// TwinCAT 3 PLC project PLC_1
// Title: ProBox
// Company: Swisslog
// Author: .
// ProjectVersion: 1.0.0
// Description: Based on BCF 1.3.0
// ProgramVersion: 3.1.4023.0
// libraries:
//   Tc2_EtherCAT, * (Beckhoff Automation GmbH)
//   Tc2_MC2, * (Beckhoff Automation GmbH)
//   Tc2_MDP, * (Beckhoff Automation GmbH)
//   Tc2_Standard, * (Beckhoff Automation GmbH)
//   Tc2_System, * (Beckhoff Automation GmbH)
//   Tc2_TcpIp, * (Beckhoff Automation GmbH)
//   Tc2_Utilities, * (Beckhoff Automation GmbH)
//   Tc3_Module, * (Beckhoff Automation GmbH)
// project tree:
//   10_Project/10_App/10_Config/00_GVLs/ Groups.TcGVL, GVL_Safety.TcGVL, HardwareMapping.TcGVL, Positions.TcGVL, ProBoxSystem.TcGVL, Subsystem.TcGVL
//   10_Project/10_App/10_Config/01_DUTs/ E_ElementNumber.TcDUT, E_FunctionNumber.TcDUT, E_GroupNumber.TcDUT
//   10_Project/10_App/10_Config/ F_ConfigCommunication.TcPOU, F_ConfigExternalDestination.TcPOU, F_ConfigGroup.TcPOU, F_ConfigGroupManager.TcPOU, F_ConfigPosition.TcPOU, F_ConfigPosition_001.TcPOU, F_ConfigPosition_002.TcPOU, F_ConfigProduct.TcPOU, F_ConfigSubSystem.TcPOU, F_UpdateISR.TcPOU, F_UpdateReferences.TcPOU
//   10_Project/10_App/11_Custom/ FB_ElementCompositionCustomized.TcPOU, FB_FunctionCompositionCustomized.TcPOU, FB_GroupCompositionCustomized.TcPOU, FB_HardwareInputs.TcPOU, FB_HardwareOutputs.TcPOU, FB_SafetyCompositionCustomized.TcPOU, FB_SubsystemCompositionCustomized.TcPOU, F_DebugCompositionCustomization.TcPOU
//   10_Project/10_App/12_FlowControl/00_GVLs/ FlowControl.TcGVL
//   10_Project/10_App/12_FlowControl/ FB_MergingService.TcPOU, FB_MergingService_001.TcPOU, FB_RoutingService.TcPOU, FB_RoutingService_001.TcPOU
//   10_Project/11_Emu/10_Config/00_GVLs/ GroupsEmulation.TcGVL, PositionsEmulation.TcGVL, SubsystemEmulation.TcGVL
//   10_Project/11_Emu/10_Config/ F_ConfigCommunicationEmulation.TcPOU, F_ConfigGroupEmulation.TcPOU, F_ConfigPositionEmulation.TcPOU, F_ConfigPositionEmulation_001.TcPOU, F_ConfigPositionEmulation_002.TcPOU, F_ConfigProductEmulation.TcPOU, F_ConfigSubSystemEmulation.TcPOU, F_UpdateReferencesEmulation.TcPOU
//   20_Product/10_BCF/10_Base/00_GVLs/ GVR_Table.TcGVL, ISR_Table.TcGVL, RegistryEmulation.TcGVL, SDI_Table.TcGVL, SDO_Table.TcGVL, System.TcGVL, SystemEmulation.TcGVL
//   20_Product/10_BCF/10_Base/01_DUTs/ E_CM_Index.TcDUT, E_CM_Mode.TcDUT, E_ErrorState.TcDUT, E_ErrorType.TcDUT, E_MFCS_Channel.TcDUT, E_PositionMode.TcDUT, E_PositionState.TcDUT, ST_Base.TcDUT, ST_CM_Base.TcDUT, ST_CM_GeneralData.TcDUT, ST_CM_Log.TcDUT, ST_CM_Settings.TcDUT, ST_ISR_Table.TcDUT, ST_PointerSet.TcDUT, ST_PositionInfo.TcDUT, ST_PositionState.TcDUT, ST_SDI_Table.TcDUT, ST_VIR_Data.TcDUT
//   20_Product/10_BCF/10_Base/10_StateMachine/ A_InstancePath.TcDUT, A_StateText.TcDUT, FB_StateMachine.TcPOU, I_StateMachineTextCallback.TcIO
//   20_Product/10_BCF/10_Base/11_Com/01_Stringhandling/ F_InstancePathRemovals.TcPOU, F_StringCopy.TcPOU, F_StringFromDatestruct.TcPOU, F_StringFromTime.TcPOU, F_StringFromTimestruct.TcPOU, F_StringFromUlint.TcPOU, F_StringFromWord.TcPOU, F_StringToTimeDate.TcPOU
//   20_Product/10_BCF/10_Base/11_Com/02_Timings/ E_BlinkFrequencies.TcDUT, F_GetBlinkCycle.TcPOU, F_GetTimeMsDiff.TcPOU, F_GetTimeMsTick.TcPOU, F_GetTimeRemain.TcPOU
//   20_Product/10_BCF/10_Base/11_Com/12_DebugMsg/00_GVLs/ DebugTextBlocks.TcGVL
//   20_Product/10_BCF/10_Base/11_Com/12_DebugMsg/01_DUTs/ E_DebugMsgType.TcDUT, ST_CFG_DebugMsgManager.TcDUT
//   20_Product/10_BCF/10_Base/11_Com/12_DebugMsg/20_TraceHandler/ FB_TraceHandler.TcPOU, I_TraceHandler.TcIO
//   20_Product/10_BCF/10_Base/11_Com/12_DebugMsg/20_TraceHandler/_internal/ A_TracePath.TcDUT (not stored)
//   20_Product/10_BCF/10_Base/11_Com/12_DebugMsg/20_TraceHandler/_internal/entry/ FB_TraceEntry.TcPOU (not stored)
//   20_Product/10_BCF/10_Base/11_Com/12_DebugMsg/20_TraceHandler/_internal/hdd_monitor/ E_ReadHddUsageStates.TcDUT (not stored), FB_HddUsage.TcPOU (not stored), F_DiskSpaceToString.TcPOU (not stored), I_HddUsage.TcIO (not stored)
//   20_Product/10_BCF/10_Base/11_Com/12_DebugMsg/20_TraceHandler/_internal/states/ E_TraceCheckStates.TcDUT (not stored), E_TraceDeleteStates.TcDUT (not stored), E_TraceHddUsageStates.TcDUT (not stored), E_TraceWriteStates.TcDUT (not stored)
//   20_Product/10_BCF/10_Base/11_Com/12_DebugMsg/20_TraceHandler/_internal/statistics/ FB_TraceHandlerStatistics.TcPOU (not stored), I_TraceHandlerStatistics.TcIO (not stored)
//   20_Product/10_BCF/10_Base/11_Com/12_DebugMsg/ FB_DebugMsg.TcPOU, FB_DebugMsgManager.TcPOU
//   20_Product/10_BCF/10_Base/11_Com/ F_InitializeCommunication.TcPOU, F_ITC_SendVIR.TcPOU, ITF_ITC.TcIO, ITF_MFCS.TcIO, ITF_MFCS_Emulation.TcIO
//   20_Product/10_BCF/10_Base/ FB_BaseObject.TcPOU, FB_BaseObjectEmulation.TcPOU, F_ExecutionTime.TcPOU, F_MemStringReplace.TcPOU
//   20_Product/10_BCF/11_Conv/09_Emulation/ MainConvEmulation.TcPOU
//   20_Product/10_BCF/11_Conv/10_Base/00_GVLs/ Conveyor.TcGVL, ExecutionTimeTable.TcGVL, Registry.TcGVL, TU_Table.TcGVL
//   20_Product/10_BCF/11_Conv/10_Base/01_DUTs/ E_ErrorConv.TcDUT, E_EtherCAT_MasterError.TcDUT, ST_ControlRequest.TcDUT, ST_DataSet.TcDUT, ST_DataSetEmulation.TcDUT, ST_Dimension.TcDUT, ST_ElementRegistryConv.TcDUT, ST_ElementRegistryConvEmulation.TcDUT, ST_ErrorDataSet.TcDUT, ST_EtherCATDeviceStates.TcDUT, ST_ExecutionTime.TcDUT, ST_ExternalDestination.TcDUT, ST_FunctionRegistryConv.TcDUT, ST_FunctionRegistryConvEmulation.TcDUT, ST_GroupRegistryConv.TcDUT, ST_GroupRegistryConvEmulation.TcDUT, ST_InitRelease.TcDUT, ST_Interlock.TcDUT, ST_Label.TcDUT, ST_LabelEmulation.TcDUT, ST_PositionIdent.TcDUT, ST_Profile.TcDUT, ST_SubSystemRegistryConv.TcDUT, ST_SubsystemRegistryConvEmulation.TcDUT, ST_TimeStamp.TcDUT, ST_TU_Data.TcDUT, ST_TU_DataEmulation.TcDUT, ST_TU_ID.TcDUT, ST_ZoneRegistryConv.TcDUT, U_ErrorCode.TcDUT
//   20_Product/10_BCF/11_Conv/10_Base/13_GroupManager/01_DUTs/ ST_CFG_GroupManager.TcDUT
//   20_Product/10_BCF/11_Conv/10_Base/13_GroupManager/ FB_GroupManager.TcPOU
//   20_Product/10_BCF/11_Conv/10_Base/ ConveyorEmulation.TcGVL, FB_CommunicationComposition.TcPOU, FB_CommunicationCompositionEmulation.TcPOU, FB_DeleteOldTU_Data.TcPOU, FB_ElementComposition.TcPOU, FB_ElementCompositionEmulation.TcPOU, FB_FunctionComposition.TcPOU, FB_FunctionCompositionEmulation.TcPOU, FB_GroupComposition.TcPOU, FB_GroupCompositionEmulation.TcPOU, FB_SubSystemComposition.TcPOU, FB_SubSystemCompositionEmulation.TcPOU, F_DeleteDestination.TcPOU, F_DeleteTU_Data.TcPOU, F_GetTU_DataIndex.TcPOU, F_GetVirtualDestination.TcPOU, F_InsertTU_Data.TcPOU, F_MonitorEtherCAT_Master.TcPOU, F_ResetError.TcPOU, F_SearchAssignmentId.TcPOU, F_SearchPositionOfTU_Index.TcPOU, F_SearchTU_ByHashCode.TcPOU, F_SetError.TcPOU
//   20_Product/10_BCF/11_Conv/11_Com/11_ITC/01_DUTs/ E_ITC_MsgTypeConv.TcDUT, ST_CFG_ITC_ManagerConv.TcDUT, ST_ITC_ADD_TU_DATA.TcDUT, ST_ITC_ATQ.TcDUT, ST_ITC_ATR.TcDUT, ST_ITC_DAQ.TcDUT, ST_ITC_DAR.TcDUT, ST_ITC_DIQ.TcDUT, ST_ITC_ECQ.TcDUT, ST_ITC_ECR.TcDUT, ST_ITC_ERQ.TcDUT, ST_ITC_ERR.TcDUT, ST_ITC_ESQ.TcDUT, ST_ITC_ESR.TcDUT, ST_ITC_FCQ.TcDUT, ST_ITC_FCR.TcDUT, ST_ITC_FSQ.TcDUT, ST_ITC_FSR.TcDUT, ST_ITC_GCQ.TcDUT, ST_ITC_GCR.TcDUT, ST_ITC_GDQ.TcDUT, ST_ITC_GDR.TcDUT, ST_ITC_GeneralData.TcDUT (not stored), ST_ITC_GSQ.TcDUT (not stored), ST_ITC_GSR.TcDUT (not stored), ST_ITC_GVQ.TcDUT (not stored), ST_ITC_GVR.TcDUT (not stored), ST_ITC_IPR.TcDUT (not stored), ST_ITC_IRQ.TcDUT (not stored), ST_ITC_ISR.TcDUT (not stored), ST_ITC_ManualMotion.TcDUT (not stored), ST_ITC_ManualMotionAxis.TcDUT (not stored), ST_ITC_ManualMotionSelection.TcDUT (not stored), ST_ITC_ManualMotionSpeed.TcDUT (not stored), ST_ITC_MCQ.TcDUT (not stored), ST_ITC_MCR.TcDUT (not stored), ST_ITC_POR.TcDUT (not stored), ST_ITC_RAA.TcDUT (not stored), ST_ITC_RAA_CommandArgs.TcDUT (not stored), ST_ITC_RAC.TcDUT (not stored), ST_ITC_RAQ.TcDUT (not stored), ST_ITC_RDQ.TcDUT (not stored), ST_ITC_RDR.TcDUT (not stored), ST_ITC_RTQ.TcDUT (not stored), ST_ITC_RTR.TcDUT (not stored), ST_ITC_SCQ.TcDUT (not stored), ST_ITC_SCR.TcDUT (not stored), ST_ITC_SDI.TcDUT (not stored), ST_ITC_SDO.TcDUT (not stored), ST_ITC_SIQ.TcDUT (not stored), ST_ITC_SIR.TcDUT (not stored), ST_ITC_SNR.TcDUT (not stored), ST_ITC_SSQ.TcDUT (not stored), ST_ITC_SSR.TcDUT (not stored), ST_ITC_TDQ.TcDUT (not stored), ST_ITC_TDR.TcDUT (not stored), ST_ITC_TTA.TcDUT (not stored), ST_ITC_TTC.TcDUT (not stored), ST_ITC_TTQ.TcDUT (not stored), ST_ITC_TUQ.TcDUT (not stored), ST_ITC_TUR.TcDUT (not stored), ST_ITC_VIQ.TcDUT (not stored), ST_ITC_VIR.TcDUT (not stored), ST_ITC_VIR_SET.TcDUT (not stored)
//   20_Product/10_BCF/11_Conv/11_Com/11_ITC/ FB_ITC_Conveyor.TcPOU, FB_ITC_ConveyorEmulation.TcPOU, F_ITC_SendATR.TcPOU, F_ITC_SendDAR.TcPOU, F_ITC_SendECR.TcPOU, F_ITC_SendERR.TcPOU, F_ITC_SendESR.TcPOU, F_ITC_SendFCR.TcPOU, F_ITC_SendFSR.TcPOU, F_ITC_SendGCR.TcPOU, F_ITC_SendGDR.TcPOU, F_ITC_SendGSR.TcPOU, F_ITC_SendGVR.TcPOU, F_ITC_SendIPR.TcPOU, F_ITC_SendISR.TcPOU, F_ITC_SendMCR.TcPOU, F_ITC_SendMSG.TcPOU, F_ITC_SendPOR.TcPOU, F_ITC_SendRAC.TcPOU, F_ITC_SendRAQ.TcPOU, F_ITC_SendRDR.TcPOU, F_ITC_SendRTR.TcPOU, F_ITC_SendSCR.TcPOU, F_ITC_SendSDI.TcPOU, F_ITC_SendSIR.TcPOU, F_ITC_SendSNR.TcPOU, F_ITC_SendSSR.TcPOU, F_ITC_SendTDR.TcPOU, F_ITC_SendTTC.TcPOU, F_ITC_SendTTQ.TcPOU, F_ITC_SendTUR.TcPOU, ITF_ITC_Emulation.TcIO
//   20_Product/10_BCF/11_Conv/11_Com/12_MFCS/11_SIS/01_DUTs/ ST_CFG_SIS_BaseDriver.TcDUT (not stored)
//   20_Product/10_BCF/11_Conv/11_Com/12_MFCS/11_SIS/11_SIS_6_0/00_GVLs/ SIS_6_0.TcGVL (not stored), SIS_6_0_Emulation.TcGVL (not stored)
//   20_Product/10_BCF/11_Conv/11_Com/12_MFCS/11_SIS/11_SIS_6_0/01_DUTs/ ST_ATQ_6_0.TcDUT (not stored), ST_ATR_6_0.TcDUT (not stored), ST_CFG_SIS_MsgManager_6_0.TcDUT (not stored), ST_DAQ_6_0.TcDUT (not stored), ST_DAR_6_0.TcDUT (not stored), ST_DIQ_6_0.TcDUT (not stored), ST_ECQ_6_0.TcDUT (not stored), ST_ECR_6_0.TcDUT (not stored), ST_ERQ_6_0.TcDUT (not stored), ST_ERR_6_0.TcDUT (not stored), ST_ESQ_6_0.TcDUT (not stored), ST_ESR_6_0.TcDUT (not stored), ST_FCQ_6_0.TcDUT (not stored), ST_FCR_6_0.TcDUT (not stored), ST_FSQ_6_0.TcDUT (not stored), ST_FSR_6_0.TcDUT (not stored), ST_GCQ_6_0.TcDUT (not stored), ST_GCR_6_0.TcDUT (not stored), ST_GDQ_6_0.TcDUT (not stored), ST_GDR_6_0.TcDUT (not stored), ST_GSQ_6_0.TcDUT (not stored), ST_GSR_6_0.TcDUT (not stored), ST_GVQ_6_0.TcDUT (not stored), ST_GVR_6_0.TcDUT (not stored), ST_IPR_6_0.TcDUT (not stored), ST_IRQ_6_0.TcDUT (not stored), ST_ISR_6_0.TcDUT (not stored), ST_MCQ_6_0.TcDUT (not stored), ST_MCR_6_0.TcDUT (not stored), ST_POR_6_0.TcDUT (not stored), ST_RAA_6_0.TcDUT (not stored), ST_RAA_6_0_CommandArgs.TcDUT (not stored), ST_RAC_6_0.TcDUT (not stored), ST_RDQ_6_0.TcDUT (not stored), ST_RDR_6_0.TcDUT (not stored), ST_RTQ_6_0.TcDUT (not stored), ST_RTR_6_0.TcDUT (not stored), ST_SCQ_6_0.TcDUT (not stored), ST_SCR_6_0.TcDUT (not stored), ST_SDI_6_0.TcDUT (not stored), ST_SDO_6_0.TcDUT (not stored), ST_SendTelegrams_6_0.TcDUT (not stored), ST_SIQ_6_0.TcDUT (not stored), ST_SIR_6_0.TcDUT (not stored), ST_SNR_6_0.TcDUT (not stored), ST_SSQ_6_0.TcDUT (not stored), ST_SSR_6_0.TcDUT (not stored), ST_TDQ_6_0.TcDUT (not stored), ST_TDR_6_0.TcDUT (not stored), ST_TTA_6_0.TcDUT (not stored), ST_TTC_6_0.TcDUT (not stored), ST_TTQ_6_0.TcDUT (not stored), ST_TUQ_6_0.TcDUT (not stored), ST_TUR_6_0.TcDUT (not stored), ST_VIQ_6_0.TcDUT (not stored), ST_VIR_6_0.TcDUT (not stored), ST_VIR_SET_6_0.TcDUT (not stored)
//   20_Product/10_BCF/11_Conv/11_Com/12_MFCS/11_SIS/11_SIS_6_0/ FB_SIS_MsgManager_6_0.TcPOU (not stored), FB_SIS_MsgManager_6_0_Emulation.TcPOU (not stored)
//   20_Product/10_BCF/11_Conv/11_Com/12_MFCS/11_SIS/12_SIS_6_1/00_GVLs/ SIS_6_1.TcGVL (not stored), SIS_6_1_Emulation.TcGVL (not stored)
//   20_Product/10_BCF/11_Conv/11_Com/12_MFCS/11_SIS/12_SIS_6_1/01_DUTs/ ST_ATQ_6_1.TcDUT (not stored), ST_ATR_6_1.TcDUT (not stored), ST_CFG_SIS_MsgManager_6_1.TcDUT (not stored), ST_DAQ_6_1.TcDUT (not stored), ST_DAR_6_1.TcDUT (not stored), ST_DIQ_6_1.TcDUT (not stored), ST_ECQ_6_1.TcDUT (not stored), ST_ECR_6_1.TcDUT (not stored), ST_ERQ_6_1.TcDUT (not stored), ST_ERR_6_1.TcDUT (not stored), ST_ESQ_6_1.TcDUT (not stored), ST_ESR_6_1.TcDUT (not stored), ST_FCQ_6_1.TcDUT (not stored), ST_FCR_6_1.TcDUT (not stored), ST_FSQ_6_1.TcDUT (not stored), ST_FSR_6_1.TcDUT (not stored), ST_GCQ_6_1.TcDUT (not stored), ST_GCR_6_1.TcDUT (not stored), ST_GDQ_6_1.TcDUT (not stored), ST_GDR_6_1.TcDUT (not stored), ST_GSQ_6_1.TcDUT (not stored), ST_GSR_6_1.TcDUT (not stored), ST_GVQ_6_1.TcDUT (not stored), ST_GVR_6_1.TcDUT (not stored), ST_IPR_6_1.TcDUT (not stored), ST_IRQ_6_1.TcDUT (not stored), ST_ISR_6_1.TcDUT (not stored), ST_MCQ_6_1.TcDUT (not stored), ST_MCR_6_1.TcDUT (not stored), ST_POR_6_1.TcDUT (not stored), ST_RAA_6_1.TcDUT (not stored), ST_RAA_6_1_CommandArgs.TcDUT (not stored), ST_RAC_6_1.TcDUT (not stored), ST_RAQ_6_1.TcDUT (not stored), ST_RDQ_6_1.TcDUT (not stored), ST_RDR_6_1.TcDUT (not stored), ST_RTQ_6_1.TcDUT (not stored), ST_RTR_6_1.TcDUT (not stored), ST_SCQ_6_1.TcDUT (not stored), ST_SCR_6_1.TcDUT (not stored), ST_SDI_6_1.TcDUT (not stored), ST_SDO_6_1.TcDUT (not stored), ST_SendTelegrams_6_1.TcDUT (not stored), ST_SIQ_6_1.TcDUT (not stored), ST_SIR_6_1.TcDUT (not stored), ST_SNR_6_1.TcDUT (not stored), ST_SSQ_6_1.TcDUT (not stored), ST_SSR_6_1.TcDUT (not stored), ST_TDQ_6_1.TcDUT (not stored), ST_TDR_6_1.TcDUT (not stored), ST_TTA_6_1.TcDUT (not stored), ST_TTC_6_1.TcDUT (not stored), ST_TTQ_6_1.TcDUT (not stored), ST_TUQ_6_1.TcDUT (not stored), ST_TUR_6_1.TcDUT (not stored), ST_VIQ_6_1.TcDUT (not stored), ST_VIR_6_1.TcDUT (not stored), ST_VIR_SET_6_1.TcDUT (not stored)
//   20_Product/10_BCF/11_Conv/11_Com/12_MFCS/11_SIS/12_SIS_6_1/ FB_SIS_MsgManager_6_1.TcPOU (not stored), FB_SIS_MsgManager_6_1_Emulation.TcPOU (not stored)
//   20_Product/10_BCF/11_Conv/11_Com/12_MFCS/11_SIS/ FB_SIS_BaseDriver.TcPOU (not stored)
//   20_Product/10_BCF/11_Conv/11_Com/13_Sub-Sub/01_DUTs/10_Config/ ST_CFG_STI_Conveyor.TcDUT (not stored)
//   20_Product/10_BCF/11_Conv/11_Com/13_Sub-Sub/01_DUTs/ ST_CFG_STI_ConveyorEmulation.TcDUT (not stored), ST_InOutputsSTI_Conveyor.TcDUT (not stored), ST_STI_Channel.TcDUT (not stored), ST_STI_ChannelEmulation.TcDUT (not stored), ST_STI_ConveyorData.TcDUT (not stored), ST_STI_ConveyorDataEmulation.TcDUT (not stored), ST_STI_Emulation.TcDUT (not stored), ST_STI_TU_Data.TcDUT (not stored)
//   20_Product/10_BCF/11_Conv/11_Com/13_Sub-Sub/12_STI_Conveyor/ FB_STI_Conveyor.TcPOU (not stored), FB_STI_ConveyorEmulation.TcPOU (not stored), FB_STI_ConveyorEmulation_V2.TcPOU (not stored), FB_STI_Conveyor_V2.TcPOU (not stored)
//   20_Product/10_BCF/11_Conv/11_Com/13_Sub-Sub/13_STI_EtherCAT/01_DUTs/ ST_CFG_STI_EtherCAT_Conveyor.TcDUT (not stored), ST_HW_InOutputsSTI_EtherCAT_Conveyor.TcDUT (not stored), ST_HW_InputsEtherCAT_Bridge.TcDUT (not stored), ST_HW_InputsEtherCAT_ConveyorInterface.TcDUT (not stored), ST_HW_OutputsEtherCAT_Bridge.TcDUT (not stored), ST_HW_OutputsEtherCAT_ConveyorInterface.TcDUT (not stored), ST_InOutputsSTI_EtherCAT_Conveyor.TcDUT (not stored), ST_STI_EtherCAT_ConveyorDataEmulation.TcDUT (not stored)
//   20_Product/10_BCF/11_Conv/11_Com/13_Sub-Sub/13_STI_EtherCAT/ FB_STI_EtherCAT_Conveyor.TcPOU (not stored), FB_STI_EtherCAT_ConveyorEmulation.TcPOU (not stored)
//   20_Product/10_BCF/11_Conv/11_Com/13_Sub-Sub/ FB_STI_SendReceiveTU_Data_6_0.TcPOU, FB_STI_SendReceiveTU_Data_6_1.TcPOU, FB_STI_SendTU_Trigger_6_0.TcPOU, FB_STI_SendTU_Trigger_6_1.TcPOU, ITF_SubsystemTransport.TcIO, ITF_SubsystemTransportEmulation.TcIO
//   20_Product/10_BCF/11_Conv/12_E_Functions/01_DUTs/ E_ActionState.TcDUT, E_ActionType.TcDUT, E_DriveDirection.TcDUT, E_FunctionType.TcDUT, E_HandOverState.TcDUT, E_ITC_FunctionControlCode.TcDUT, E_Signalstate.TcDUT, E_SpeedControlState.TcDUT, E_TakeoverSignalstate.TcDUT, E_TakeOverState.TcDUT, E_TransportState.TcDUT, E_TUR_SendModes.TcDUT, ST_AddOn.TcDUT, ST_AddOnData.TcDUT, ST_AddonEntry.TcDUT, ST_AddOnOrders.TcDUT, ST_AddOnResult.TcDUT, ST_CFG_Function.TcDUT, ST_CFG_FunctionLink.TcDUT, ST_CFG_Zone.TcDUT, ST_CM_ZoneBase.TcDUT, ST_FunctionBase.TcDUT, ST_FunctionData.TcDUT, ST_FunctionElement.TcDUT, ST_FunctionErrorStruct.TcDUT, ST_FunctionInterface.TcDUT, ST_FunctionInterfaceIn.TcDUT, ST_FunctionInterfaceOut.TcDUT, ST_FunctionMemberList.TcDUT, ST_FunctionOrders.TcDUT, ST_ITC_Function.TcDUT, ST_ITC_FunctionCommands.TcDUT, ST_ITC_FunctionITC.TcDUT, ST_ITC_Zone.TcDUT, ST_ITC_ZoneCommands.TcDUT, ST_ITC_ZoneFlags.TcDUT, ST_LastTUdata.TcDUT, ST_TransportControlData.TcDUT, ST_TransportControlParam.TcDUT, ST_TransportControl_Inputs.TcDUT, ST_TransportControl_Outputs.TcDUT, ST_TransportData.TcDUT, ST_TransportDataRequest.TcDUT, ST_TransportEnable.TcDUT, ST_TransportParam.TcDUT, ST_ZoneData.TcDUT, ST_ZoneErrorStruct.TcDUT, ST_ZoneInterface.TcDUT, ST_ZoneInterfaceIn.TcDUT, ST_ZoneInterfaceOut.TcDUT
//   20_Product/10_BCF/11_Conv/12_E_Functions/09_Emulation/01_DUTs/ E_TransportControlAddTU_Emulation.TcDUT (not stored), E_TransportControlRemoveTU_Emulation.TcDUT (not stored), E_TransportDirection.TcDUT (not stored), ST_CFG_FunctionEmulation.TcDUT (not stored), ST_FunctionBaseEmulation.TcDUT (not stored), ST_FunctionDataEmulation.TcDUT (not stored), ST_ITC_FunctionCommandsEmulation.TcDUT (not stored), ST_ITC_FunctionEmulation.TcDUT (not stored), ST_ITC_FunctionITC_Emulation.TcDUT (not stored), ST_ITC_ZoneCommandsEmulation.TcDUT (not stored), ST_ITC_ZoneEmulation.TcDUT (not stored), ST_SetHW_Inputs.TcDUT (not stored), ST_TransportControlDataEmulation.TcDUT (not stored), ST_TransportControlParamEmulation.TcDUT (not stored), ST_TransportDataEmulation.TcDUT (not stored), ST_TransportParamEmulation.TcDUT (not stored), ST_ZoneDataEmulation.TcDUT (not stored)
//   20_Product/10_BCF/11_Conv/12_E_Functions/09_Emulation/10_Helper/ FB_HandoverEmulation.TcPOU (not stored), FB_TakeoverEmulation.TcPOU (not stored), FB_TransportControlEmulation.TcPOU (not stored), F_CreateEmulationTU_DataString.TcPOU (not stored), F_GetAdjacentTransportDataEmulation.TcPOU (not stored), F_GetAllZoneDataEmulation.TcPOU (not stored), F_GetFunctionDataEmulation.TcPOU (not stored), F_GetTransportControlDataEmulation.TcPOU (not stored), F_GetTU_DataIndexEmulation.TcPOU (not stored), F_GetTU_PresentStateEmulation.TcPOU (not stored), F_GetZoneDataEmulation.TcPOU (not stored), F_InsertTU_DataEmulation.TcPOU (not stored), F_MoveTU_DataIndexEmulation.TcPOU (not stored), F_SetZoneOccupiedEmulation.TcPOU (not stored), I_HandoverEmulationListener.TcIO (not stored), I_TakeoverEmulationListener.TcIO (not stored)
//   20_Product/10_BCF/11_Conv/12_E_Functions/09_Emulation/ FB_FunctionConvEmulation.TcPOU
//   20_Product/10_BCF/11_Conv/12_E_Functions/10_Helper/01_DUTs/ E_HandoverTrackingState.TcDUT (not stored), E_TakeoverTrackingMergeState.TcDUT (not stored), E_TakeoverTrackingState.TcDUT (not stored)
//   20_Product/10_BCF/11_Conv/12_E_Functions/10_Helper/02_ITFs/ I_HandoverListener.TcIO (not stored), I_TakeoverListener.TcIO (not stored)
//   20_Product/10_BCF/11_Conv/12_E_Functions/10_Helper/10_Slugging/ E_SluggingAddOnDirections.TcDUT (not stored), FB_SluggingAddOn.TcPOU (not stored), FB_SluggingAddOnEmulation.TcPOU (not stored), I_SluggingAddOn.TcIO (not stored)
//   20_Product/10_BCF/11_Conv/12_E_Functions/10_Helper/10_Slugging/sensor_emulation/ E_SensorEmulateModes.TcTLEO (not stored), FB_EmulateSensor.TcPOU (not stored), F_EmptyZoneData.TcPOU (not stored), F_InRangeDint.TcPOU (not stored), F_IsValidFunctionNumber.TcPOU (not stored)
//   20_Product/10_BCF/11_Conv/12_E_Functions/10_Helper/10_Slugging/summary/ FB_SluggingAddOn_Summary.TcPOU (not stored), I_SluggingAddOn_Summary.TcIO (not stored)
//   20_Product/10_BCF/11_Conv/12_E_Functions/10_Helper/10_Slugging/_internal/ E_SluggingAddOnStates.TcDUT (not stored), ST_SluggingAddOnOrder_Zone.TcDUT (not stored), ST_SluggingAddOn_Config.TcDUT (not stored), ST_SluggingAddOn_Zone.TcDUT (not stored)
//   20_Product/10_BCF/11_Conv/12_E_Functions/10_Helper/ FB_DistanceMeter.TcPOU, FB_GetDistance.TcPOU, FB_GetEncoderResolution.TcPOU, FB_Handover.TcPOU, FB_HandoverTracking.TcPOU, FB_HandoverTrackingDivert.TcPOU, FB_SpeedControl.TcPOU, FB_SpeedControlRamp.TcPOU, FB_Takeover.TcPOU, FB_TakeoverTracking.TcPOU, FB_TakeoverTrackingMerge.TcPOU, FB_TransportControl.TcPOU, F_AckAddon.TcPOU, F_AddDividerToSisString.TcPOU, F_CheckDestination.TcPOU, F_CheckSubsystem.TcPOU, F_CreateTU_DataString.TcPOU, F_EqualSisNames.TcPOU, F_FindElement.TcPOU, F_FindFunction.TcPOU, F_FindGroup.TcPOU, F_GetAdjacentTransportData.TcPOU, F_GetDestination.TcPOU, F_GetFunctionErrorData.TcPOU, F_GetFunctionExternalErrorData.TcPOU, F_GetFunctionInterface.TcPOU, F_GetFunctionInterlock.TcPOU, F_GetFunctionName.TcPOU, F_GetFunctionOperationState.TcPOU, F_GetFunctionSettings.TcPOU, F_GetFunctionType.TcPOU, F_GetNumberOfZones.TcPOU, F_GetTransportControlData.TcPOU, F_GetZoneData.TcPOU, F_GetZoneErrorData.TcPOU, F_GetZoneExternErrorData.TcPOU, F_GetZoneInterface.TcPOU, F_GetZonesCount.TcPOU, F_GetZonesData.TcPOU, F_GetZonesInterface.TcPOU, F_InitializeAllFunctions.TcPOU, F_InitializeFunction.TcPOU, F_IsFunctionErrorPending.TcPOU, F_IsFunctionInitialized.TcPOU, F_MoveTU_DataIndex.TcPOU, F_ResetExternalFunctionError.TcPOU, F_ResetFunctionError.TcPOU, F_SearchFunctionPosition.TcPOU, F_SetEnableHandOver.TcPOU, F_SetEnableTakeOver.TcPOU, F_SetEnableTransport.TcPOU, F_SetExternalFunctionError.TcPOU, F_StoppingDistance.TcPOU
//   20_Product/10_BCF/11_Conv/12_E_Functions/ FB_FunctionConv.TcPOU
//   20_Product/10_BCF/11_Conv/13_Elements/01_DUTs/ E_ElementType.TcDUT, E_ITC_ElementControlCode.TcDUT, ST_CFG_Element.TcDUT, ST_ElementBase.TcDUT, ST_ElementData.TcDUT, ST_ElementErrorStruct.TcDUT, ST_ElementInterface.TcDUT, ST_ElementInterfaceIn.TcDUT, ST_ElementInterfaceOut.TcDUT, ST_ElementMasterSlave.TcDUT, ST_ElementMasterSlaveEntry.TcDUT, ST_ElementMemberList.TcDUT, ST_ElementState.TcDUT, ST_FunctionEntry.TcDUT, ST_ITC_Element.TcDUT, ST_ITC_ElementCommands.TcDUT, ST_MasterSlaveStates.TcDUT
//   20_Product/10_BCF/11_Conv/13_Elements/09_Emulation/01_DUTs/ ST_ElementBaseEmulation.TcDUT (not stored), ST_ElementDataEmulation.TcDUT (not stored), ST_ITC_ElementCommandsEmulation.TcDUT (not stored), ST_ITC_ElementEmulation.TcDUT (not stored)
//   20_Product/10_BCF/11_Conv/13_Elements/09_Emulation/ FB_ElementConvEmulation.TcPOU
//   20_Product/10_BCF/11_Conv/13_Elements/10_Helper/ F_GetElementErrorData.TcPOU, F_GetElementExternErrorData.TcPOU, F_GetElementInterface.TcPOU, F_GetElementOperationState.TcPOU, F_GetElementOrders.TcPOU, F_GetElementSettings.TcPOU, F_InitializeAllElements.TcPOU, F_InitializeElement.TcPOU, F_IsElementErrorPending.TcPOU, F_IsElementInitialized.TcPOU, F_ResetElementError.TcPOU, F_ResetExternalElementError.TcPOU, F_SearchElementPosition.TcPOU, F_SetExternalElementError.TcPOU
//   20_Product/10_BCF/11_Conv/13_Elements/ FB_ElementConv.TcPOU
//   20_Product/10_BCF/11_Conv/14_Groups/01_DUTs/ E_GroupType.TcDUT, E_ITC_GroupControlCode.TcDUT, ST_CFG_Group.TcDUT, ST_GroupBase.TcDUT, ST_GroupData.TcDUT, ST_GroupErrorStruct.TcDUT, ST_GroupInterface.TcDUT, ST_GroupInterfaceIn.TcDUT, ST_GroupInterfaceOut.TcDUT, ST_GroupManagerElementMember.TcDUT, ST_GroupManagerGroupMember.TcDUT, ST_ITC_Group.TcDUT, ST_ITC_GroupCommands.TcDUT, ST_ITC_GroupEmulation.TcDUT
//   20_Product/10_BCF/11_Conv/14_Groups/09_Emulation/01_DUTs/ ST_GroupBaseEmulation.TcDUT (not stored), ST_GroupDataEmulation.TcDUT (not stored), ST_ITC_GroupCommandsEmulation.TcDUT (not stored)
//   20_Product/10_BCF/11_Conv/14_Groups/09_Emulation/ FB_GroupConvEmulation.TcPOU
//   20_Product/10_BCF/11_Conv/14_Groups/10_Helper/ F_GetGroupErrorData.TcPOU, F_GetGroupExternErrorData.TcPOU, F_GetGroupInterface.TcPOU, F_GetGroupName.TcPOU, F_GetGroupOperationState.TcPOU, F_GetGroupSettings.TcPOU, F_InitializeAllGroups.TcPOU, F_InitializeGroup.TcPOU, F_IsGroupInitialized.TcPOU, F_ResetExternalGroupError.TcPOU, F_ResetGroupError.TcPOU, F_SearchGroupNumber.TcPOU, F_SetExternalGroupError.TcPOU
//   20_Product/10_BCF/11_Conv/14_Groups/ FB_GroupConv.TcPOU
//   20_Product/10_BCF/11_Conv/15_Subsystem/01_DUTs/ E_ITC_SubSystemControlCode.TcDUT, E_SystemInfo.TcDUT, ST_ITC_SubSystem.TcDUT, ST_ITC_SubSystemCommands.TcDUT, ST_SubSystemBase.TcDUT, ST_SubSystemData.TcDUT, ST_SubSystemErrorStruct.TcDUT, ST_SubSystemInterface.TcDUT, ST_SubSystemInterfaceIn.TcDUT, ST_SubSystemInterfaceOut.TcDUT
//   20_Product/10_BCF/11_Conv/15_Subsystem/09_Emulation/01_DUTs/ ST_ITC_SubSystemCommandsEmulation.TcDUT (not stored), ST_ITC_SubSystemEmulation.TcDUT (not stored), ST_SubsystemBaseEmulation.TcDUT (not stored), ST_SubSystemDataEmulation.TcDUT (not stored)
//   20_Product/10_BCF/11_Conv/15_Subsystem/09_Emulation/ FB_SubsystemConvEmulation.TcPOU
//   20_Product/10_BCF/11_Conv/15_Subsystem/10_Helper/ F_GetSubSystemErrorData.TcPOU, F_GetSubSystemExternErrorData.TcPOU, F_GetSubSystemInterface.TcPOU, F_GetSubsystemOperationState.TcPOU, F_GetSubSystemSettings.TcPOU, F_InitializeSubsystem.TcPOU, F_IsSubsystemInitialized.TcPOU, F_ResetExternalSubsystemError.TcPOU, F_ResetSubsystemError.TcPOU, F_SetExternalSubsystemError.TcPOU
//   20_Product/10_BCF/11_Conv/15_Subsystem/11_DummySubsystem/01_DUTs/ ST_CFG_DummySubsystem.TcDUT (not stored), ST_CFG_Subsystem.TcDUT (not stored), ST_HW_InputsSubSystemManager.TcDUT (not stored), ST_HW_OutputsSubSystemManager.TcDUT (not stored), ST_InputsSubSystemManager.TcDUT (not stored), ST_OutputsSubSystemManager.TcDUT (not stored)
//   20_Product/10_BCF/11_Conv/15_Subsystem/ FB_SubsystemConv.TcPOU
//   20_Product/10_BCF/11_Conv/ MainConv.TcPOU
//   20_Product/10_BCF/ BCF_Version.TcTLO
//   20_Product/20_ProBox/10_Base/00_GVLs/ PBTransportCtrl.TcGVL, ProBox_Conveyor.TcGVL
//   20_Product/20_ProBox/10_Base/01_DUTs/ E_ErrorProduct.TcDUT
//   20_Product/20_ProBox/10_Base/09_Overrides/ FB_PB_FunctionConv.TcPOU, FB_PB_ITC_Conveyor.TcPOU
//   20_Product/20_ProBox/22_ProMove/01_DUTs/ASI/ ST_ASI_HW_Input.TcDUT, ST_ASI_HW_IO.TcDUT, ST_ASI_HW_Output.TcDUT, ST_HW_InputsASi_16_31.TcDUT, ST_HW_InputsASi_1_15.TcDUT, ST_HW_OutputsASi_16_31.TcDUT, ST_HW_OutputsASi_1_15.TcDUT
//   20_Product/20_ProBox/22_ProMove/01_DUTs/ E_Axis_Orientation.TcDUT, E_ProBoxMotorSpeed.TcDUT
//   20_Product/20_ProBox/22_ProMove/03_Controls/02_TransportControl/01_DUTs/ ST_CtrlInPbTc.TcDUT (not stored), ST_PB_TransportCtrl.TcDUT (not stored)
//   20_Product/20_ProBox/22_ProMove/03_Controls/02_TransportControl/ FB_PB_TransportControlEmulation.TcPOU, FB_ProBoxTransportControl.TcPOU
//   20_Product/20_ProBox/22_ProMove/03_Controls/03_SpeedControl/10_App/ FB_ProBoxSpeedControl.TcPOU (not stored)
//   20_Product/20_ProBox/22_ProMove/03_Controls/04_MotorControl/10_App/01_DUTs/ E_ProBoxMotorDirection.TcDUT (not stored)
//   20_Product/20_ProBox/22_ProMove/03_Controls/04_MotorControl/10_App/ FB_ProBoxMotorControl.TcPOU (not stored)
//   20_Product/20_ProBox/22_ProMove/03_Controls/04_MotorControl/11_Emu/ FB_MotorControlEmulation.TcPOU (not stored)
//   20_Product/20_ProBox/22_ProMove/03_Controls/05_LiftControl/10_App/01_DUTs/ E_Positions_LiftControl.TcDUT (not stored), E_States_LiftControl.TcDUT (not stored)
//   20_Product/20_ProBox/22_ProMove/03_Controls/05_LiftControl/10_App/ FB_LiftControl.TcPOU (not stored)
//   20_Product/20_ProBox/22_ProMove/03_Controls/05_LiftControl/11_Emu/ FB_LiftControlEmulation.TcPOU (not stored)
//   20_Product/20_ProBox/22_ProMove/03_Controls/06_LowLiftControl/10_App/01_DUTs/ E_Positions_LowLiftControl.TcDUT (not stored), E_States_LowLiftControl.TcDUT (not stored)
//   20_Product/20_ProBox/22_ProMove/03_Controls/06_LowLiftControl/10_App/ FB_LowLiftControl.TcPOU (not stored)
//   20_Product/20_ProBox/22_ProMove/03_Controls/06_LowLiftControl/11_Emu/ FB_LowLiftControlEmulation.TcPOU (not stored)
//   20_Product/20_ProBox/22_ProMove/03_Controls/07_TurnControl/10_App/01_DUTs/ E_Positions_TurnControl.TcDUT (not stored), E_States_TurnControl.TcDUT (not stored)
//   20_Product/20_ProBox/22_ProMove/03_Controls/07_TurnControl/10_App/ FB_TurnControl.TcPOU (not stored)
//   20_Product/20_ProBox/22_ProMove/03_Controls/07_TurnControl/11_Emu/ FB_TurnControlEmulation.TcPOU (not stored)
//   20_Product/20_ProBox/22_ProMove/03_Controls/08_StackerLiftControl/10_App/01_DUTs/ E_StackerLiftPositions.TcDUT (not stored), E_StackerLiftStates.TcDUT (not stored), ST_StackerLiftManualInp.TcDUT (not stored), ST_StackerLiftSensorInp.TcDUT (not stored)
//   20_Product/20_ProBox/22_ProMove/03_Controls/08_StackerLiftControl/10_App/ FB_StackerLiftControl.TcPOU (not stored)
//   20_Product/20_ProBox/22_ProMove/03_Controls/08_StackerLiftControl/11_Emu/ FB_StackerLiftControlEmulation.TcPOU (not stored)
//   20_Product/20_ProBox/22_ProMove/03_Controls/09_StackerForkControl/10_App/01_DUTs/ E_StackerForkPosition.TcDUT (not stored), E_StackerForkStates.TcDUT (not stored)
//   20_Product/20_ProBox/22_ProMove/03_Controls/09_StackerForkControl/10_App/ FB_StackerForkControl.TcPOU (not stored)
//   20_Product/20_ProBox/22_ProMove/03_Controls/09_StackerForkControl/11_Emu/ FB_StackerForkControlEmulation.TcPOU (not stored)
//   20_Product/20_ProBox/22_ProMove/03_Controls/10_HorizontalMotorControl/10_App/01_DUTs/ E_Positions_HorizontalControl.TcDUT (not stored), E_States_HorizontalControl.TcDUT (not stored)
//   20_Product/20_ProBox/22_ProMove/03_Controls/10_HorizontalMotorControl/10_App/ FB_HorizontalControl.TcPOU (not stored)
//   20_Product/20_ProBox/22_ProMove/03_Controls/10_HorizontalMotorControl/11_Emu/ FB_HorizontalControlEmulation.TcPOU (not stored)
//   20_Product/20_ProBox/22_ProMove/03_Controls/12_MotionPickAndDeposit/00_GVLs/ GVL_MPD.TcGVL (not stored)
//   20_Product/20_ProBox/22_ProMove/03_Controls/12_MotionPickAndDeposit/01_DUTs/ E_MotionPD_Type.TcDUT (not stored), E_MPD_CvStates.TcDUT (not stored), E_MPD_States.TcDUT (not stored), E_PickupDepositSide.TcDUT (not stored), ST_AutoAdjustVcHeight.TcDUT (not stored), ST_CFG_MotionPickupDeposit.TcDUT (not stored), ST_CFG_MPD_Drive.TcDUT (not stored), ST_CFG_PDs.TcDUT (not stored), ST_CtrlInMPD_Control.TcDUT (not stored), ST_CtrlOutMPD_Control.TcDUT (not stored), ST_EncoderHoming.TcDUT (not stored), ST_HW_InputsManControl.TcDUT (not stored), ST_HW_InputsManControlConv.TcDUT (not stored), ST_HW_InputsMPD.TcDUT (not stored), ST_HW_InputsMPD_Conv.TcDUT (not stored), ST_HW_OutputsMPD.TcDUT (not stored), ST_MPD.TcDUT (not stored), ST_MPD_CV.TcDUT (not stored), ST_MPD_SemiDriveControl.TcDUT (not stored), ST_PrioFunctions.TcDUT (not stored)
//   20_Product/20_ProBox/22_ProMove/03_Controls/12_MotionPickAndDeposit/01_DUTs/MoviDrive/ E_DriveMoverInverterType.TcDUT (not stored), E_MoveAbsoluteMode.TcDUT (not stored), E_PositioningState.TcDUT (not stored), ST_ABBDriveCtrlWord.TcDUT (not stored), ST_ABBDriveStatusWord.TcDUT (not stored), ST_MoviDriveCtrlWord.TcDUT (not stored), ST_MoviDriveManual.TcDUT (not stored), ST_MoviDriveStatusWord.TcDUT (not stored), ST_ParametersDrive.TcDUT (not stored), ST_PDO_DriveIn.TcDUT (not stored), ST_PDO_DriveOut.TcDUT (not stored), ST_SemiDriveControl.TcDUT (not stored)
//   20_Product/20_ProBox/22_ProMove/03_Controls/12_MotionPickAndDeposit/ FB_DriveMover.TcPOU, FB_EntryReqControl.TcPOU, FB_MPD_Control.TcPOU, FB_MPD_PriorityControl.TcPOU
//   20_Product/20_ProBox/22_ProMove/03_Controls/13_ExtendedRunControl/01_DUTs/ ST_CFG_ExtendedRun.TcDUT (not stored)
//   20_Product/20_ProBox/22_ProMove/03_Controls/13_ExtendedRunControl/ FB_ExtendedRun.TcPOU
//   20_Product/20_ProBox/22_ProMove/03_Controls/14_LiftTableControl/10_App/ FB_TableLiftControl.TcPOU (not stored)
//   20_Product/20_ProBox/22_ProMove/03_Controls/14_TiltControl/10_App/01_DUTs/ E_Positions_TiltControl.TcDUT (not stored), E_States_TiltControl.TcDUT (not stored)
//   20_Product/20_ProBox/22_ProMove/03_Controls/14_TiltControl/10_App/ FB_TiltControl.TcPOU (not stored)
//   20_Product/20_ProBox/22_ProMove/03_Controls/14_TiltControl/11_Emu/01_DUTs/ ST_CFG_TiltPositionEmu.TcDUT (not stored)
//   20_Product/20_ProBox/22_ProMove/03_Controls/14_TiltControl/11_Emu/ FB_TiltControlEmulation.TcPOU (not stored)
//   20_Product/20_ProBox/22_ProMove/03_Controls/15_OverhangSensorControl/10_App/ FB_OH_SensorControl.TcPOU (not stored), F_IsFwdDriveDirection.TcPOU (not stored)
//   20_Product/20_ProBox/22_ProMove/03_Controls/15_OverhangSensorControl/11_Emu/ F_OH_SensorControlEmu.TcPOU (not stored)
//   20_Product/20_ProBox/22_ProMove/03_Controls/ FB_ProBoxToElementState.TcPOU, F_ProBoxToFunctionOrders.TcPOU
//   20_Product/20_ProBox/22_ProMove/11_Addons/23_PalletMagazineAddon/10_App/01_DUTs/ ST_CFG_PalletMagazine.TcDUT (not stored), ST_CtrlInPalletmagazine.TcDUT (not stored), ST_HW_InputsPalletMagazine.TcDUT (not stored), ST_HW_OutputsPalletMagazine.TcDUT (not stored), ST_InputsPalletMagazine.TcDUT (not stored), ST_OutputsPalletMagazine.TcDUT (not stored)
//   20_Product/20_ProBox/22_ProMove/11_Addons/23_PalletMagazineAddon/10_App/ FB_PalletMagazineAddon.TcPOU (not stored)
//   20_Product/20_ProBox/22_ProMove/11_Addons/23_PalletMagazineAddon/11_Emu/01_DUTs/ ST_CFG_PalletMagazineEmulation.TcDUT (not stored)
//   20_Product/20_ProBox/22_ProMove/11_Addons/23_PalletMagazineAddon/11_Emu/ FB_PalletMagazineAddonEmulation.TcPOU (not stored)
//   20_Product/20_ProBox/22_ProMove/11_Addons/24_LoadStackerAddon/10_App/01_DUTs/ ST_CFG_Loadstacker.TcDUT (not stored), ST_CtrlInLoadstacker.TcDUT (not stored), ST_HW_InputsLoadstacker.TcDUT (not stored), ST_HW_OutputLoadStacker.TcDUT (not stored), ST_InputsLoadstacker.TcDUT (not stored), ST_LS_CfgLiftEncoder.TcDUT (not stored), ST_LS_CfgLiftEncPreset.TcDUT (not stored), ST_OutputsLoadstacker.TcDUT (not stored)
//   20_Product/20_ProBox/22_ProMove/11_Addons/24_LoadStackerAddon/10_App/01_DUTs_Base/ E_LSPM_ForkPos.TcDUT (not stored), E_LSPM_LiftPos.TcDUT (not stored), E_LSPM_LiftType.TcDUT (not stored), E_LSPM_MachineType.TcDUT (not stored), E_LSPM_Mode.TcDUT (not stored), E_LSPM_States.TcDUT (not stored), ST_LSPM_Base.TcDUT (not stored), ST_LSPM_CtrlOut.TcDUT (not stored), ST_LSPM_Inp_Element.TcDUT (not stored), ST_LSPM_Inp_ForkSensors.TcDUT (not stored), ST_LSPM_Inp_LiftSensors.TcDUT (not stored), ST_LSPM_Inp_ManualControl.TcDUT (not stored), ST_LSPM_LiftEncPos.TcDUT (not stored), ST_LSPM_OpRecover.TcDUT (not stored), ST_LSPM_Outp_Fork.TcDUT (not stored), ST_LSPM_Outp_Lift.TcDUT (not stored), ST_LSPM_States.TcDUT (not stored)
//   20_Product/20_ProBox/22_ProMove/11_Addons/24_LoadStackerAddon/10_App/ FB_LoadstackerAddon.TcPOU (not stored), FB_LSPM_Base.TcPOU (not stored)
//   20_Product/20_ProBox/22_ProMove/11_Addons/24_LoadStackerAddon/11_Emu/01_DUTs/ ST_CFG_LoadstackerAddonEmulation.TcDUT (not stored)
//   20_Product/20_ProBox/22_ProMove/11_Addons/24_LoadStackerAddon/11_Emu/ FB_LoadstackerAddonEmulation.TcPOU (not stored), FB_LS_Emu_PalletCounter.TcPOU (not stored)
//   20_Product/20_ProBox/22_ProMove/11_Addons/27_CraneXoverAddon/10_App/01_DUTs/ E_Conveyor_InterfaceState.TcDUT (not stored), E_CraneCommunicationType.TcDUT (not stored), E_CvCraneHandlerType.TcDUT (not stored), E_CvCraneXoverType.TcDUT (not stored), ST_CFG_CraneXover.TcDUT (not stored), ST_CFG_MotorTransfer.TcDUT (not stored), ST_Conveyor_Interface_5_1.TcDUT (not stored), ST_Conveyor_Interface_5_1_TU.TcDUT (not stored), ST_CraneXOverCommunication.TcDUT (not stored), ST_CtrlInCraneXover.TcDUT (not stored), ST_CtrlOutCraneXover.TcDUT (not stored), ST_HW_InputsCraneXover.TcDUT (not stored), ST_HW_InputsMotorTransfer.TcDUT (not stored), ST_HW_OutputsCraneXover.TcDUT (not stored), ST_InputsCraneXover.TcDUT (not stored), ST_MotorDriver.TcDUT (not stored), ST_OutputsCraneXover.TcDUT (not stored)
//   20_Product/20_ProBox/22_ProMove/11_Addons/27_CraneXoverAddon/10_App/ FB_CraneXoverAddon.TcPOU (not stored), FB_Crane_CV_StateHandler.TcPOU (not stored), FB_PlcCraneTcpIpCom.TcPOU (not stored)
//   20_Product/20_ProBox/22_ProMove/11_Addons/27_CraneXoverAddon/11_Emu/ FB_CraneXoverAddonEmulation.TcPOU (not stored)
//   20_Product/20_ProBox/22_ProMove/11_Addons/28_MovableStopAddon/10_App/01_DUTs/ E_DirectionMovableStop.TcDUT (not stored), E_MovableStopStates.TcDUT (not stored), ST_CFG_MovableStop.TcDUT (not stored), ST_CtrlInMovableStop.TcDUT (not stored), ST_CtrlOutMovableStop.TcDUT (not stored), ST_HW_InputsMovableStop.TcDUT (not stored), ST_HW_OutputsMovableStop.TcDUT (not stored), ST_InputsMovableStop.TcDUT (not stored), ST_MovableStopStates.TcDUT (not stored), ST_OutputsMovableStop.TcDUT (not stored)
//   20_Product/20_ProBox/22_ProMove/11_Addons/28_MovableStopAddon/10_App/ FB_MovableStopAddon.TcPOU (not stored)
//   20_Product/20_ProBox/22_ProMove/11_Addons/28_MovableStopAddon/11_Emu/01_DUTs/ ST_CFG_MovableStopAddonEmulation.TcDUT (not stored)
//   20_Product/20_ProBox/22_ProMove/11_Addons/28_MovableStopAddon/11_Emu/ FB_MovableStopAddonEmulation.TcPOU (not stored)
//   20_Product/20_ProBox/22_ProMove/11_Addons/29_FastDoor/10_App/01_DUTs/ E_DoorPos.TcDUT (not stored), E_FastDoorControlStates.TcDUT (not stored), E_FastDoorState.TcDUT (not stored), ST_CFG_FastDoor.TcDUT (not stored), ST_FastDoorData.TcDUT (not stored), ST_FastDoorStates.TcDUT (not stored), ST_HW_InputsFastDoor.TcDUT (not stored), ST_HW_OutputsFastDoor.TcDUT (not stored), ST_InputsFastDoor.TcDUT (not stored), ST_OutputsFastDoor.TcDUT (not stored)
//   20_Product/20_ProBox/22_ProMove/11_Addons/29_FastDoor/10_App/ FB_FastDoorAddon.TcPOU (not stored)
//   20_Product/20_ProBox/22_ProMove/11_Addons/29_FastDoor/11_Emu/ FB_FastDoorAddonEmulation.TcPOU (not stored)
//   20_Product/20_ProBox/22_ProMove/11_Addons/81_LiftTableAddon/10_App/01_DUTs/ E_LiftTableState.TcDUT (not stored), ST_CFG_LiftTable.TcDUT (not stored), ST_HW_InputsLiftTable.TcDUT (not stored), ST_HW_OutputsLiftTable.TcDUT (not stored), ST_InputsLiftTable.TcDUT (not stored), ST_LiftTableStates.TcDUT (not stored), ST_LiftTable_Inp_LiftSensors.TcDUT (not stored), ST_LiftTable_Inp_OP.TcDUT (not stored), ST_OutputsLiftTable.TcDUT (not stored)
//   20_Product/20_ProBox/22_ProMove/11_Addons/81_LiftTableAddon/10_App/ FB_LiftTableAddon.TcPOU (not stored)
//   20_Product/20_ProBox/22_ProMove/11_Addons/81_LiftTableAddon/11_Emu/01_DUTs/ ST_CFG_LiftTableEmulation.TcDUT (not stored)
//   20_Product/20_ProBox/22_ProMove/11_Addons/81_LiftTableAddon/11_Emu/ FB_LiftTableAddonEmulation.TcPOU (not stored)
//   20_Product/20_ProBox/22_ProMove/11_Addons/82_InOutFeedAddon/10_App/01_DUTs/ E_InOutFeedState.TcDUT (not stored), ST_CFG_InOutFeed.TcDUT (not stored), ST_CtrlInInOutFeed.TcDUT (not stored), ST_CtrlOutInOutFeed.TcDUT (not stored), ST_HW_InputsInOutFeed.TcDUT (not stored), ST_HW_OutputsInOutFeed.TcDUT (not stored), ST_InOutFeedData.TcDUT (not stored), ST_InOutFeedStates.TcDUT (not stored), ST_InputsInOutFeed.TcDUT (not stored), ST_OutputsInOutFeed.TcDUT (not stored)
//   20_Product/20_ProBox/22_ProMove/11_Addons/82_InOutFeedAddon/10_App/ FB_InOutFeedAddon.TcPOU (not stored)
//   20_Product/20_ProBox/22_ProMove/11_Addons/82_InOutFeedAddon/11_Emu/ FB_InOutFeedAddonEmulation.TcPOU (not stored)
//   20_Product/20_ProBox/22_ProMove/11_Addons/90_ProfileCheckAddon/10_App/01_DUTs/ E_LightgridType.TcDUT (not stored), E_ProfileCheckMeasurement.TcDUT (not stored), E_ProfileCheckState.TcDUT (not stored), E_ReadBeamDataState.TcDUT (not stored), ST_CFG_ProfileCheck.TcDUT (not stored), ST_CFG_ProfileRule.TcDUT (not stored), ST_CFG_SingelSensor.TcDUT (not stored), ST_CtrlInProfileCheck.TcDUT (not stored), ST_CtrlOutProfileCheck.TcDUT (not stored), ST_HW_InputsProfileCheck.TcDUT (not stored), ST_HW_OutputsProfileCheck.TcDUT (not stored), ST_InputsProfileCheck.TcDUT (not stored), ST_OutputsProfileCheck.TcDUT (not stored), ST_ProfileCheckStates.TcDUT (not stored)
//   20_Product/20_ProBox/22_ProMove/11_Addons/90_ProfileCheckAddon/10_App/ FB_ProfileCheckAddon.TcPOU (not stored), FB_ProfileCheckMeasure.TcPOU (not stored), F_ProfileCheckSensorConverter.TcPOU (not stored)
//   20_Product/20_ProBox/22_ProMove/11_Addons/90_ProfileCheckAddon/11_Emu/01_DUTs/ ST_CFG_ProfileCheckAddonEmulation.TcDUT (not stored)
//   20_Product/20_ProBox/22_ProMove/11_Addons/90_ProfileCheckAddon/11_Emu/ FB_ProfileCheckAddonEmulation.TcPOU (not stored)
//   20_Product/20_ProBox/22_ProMove/11_Addons/91_SickScannerAddon/10_App/01_DUTs/ ST_CFG_SickScanner.TcDUT (not stored), ST_CtrlInSickScanner.TcDUT (not stored), ST_CtrlOutSickScanner.TcDUT (not stored), ST_HW_InputsSickScanner.TcDUT (not stored), ST_HW_InputsSickScanner_CLV690.TcDUT (not stored), ST_HW_OutputsSickScanner.TcDUT (not stored), ST_HW_OutputsSickScanner_CLV690.TcDUT (not stored), ST_InputsSickScanner.TcDUT (not stored), ST_InputsSickScanner_CLV690.TcDUT (not stored), ST_OutputsSickScanner.TcDUT (not stored)
//   20_Product/20_ProBox/22_ProMove/11_Addons/91_SickScannerAddon/10_App/01_DUTs_Base/ E_SickScannerState.TcDUT (not stored), GVL_SickScanner.TcGVL (not stored), ITF_PB_ScannerAddon.TcIO (not stored), ST_ScannerLabelData.TcDUT (not stored), ST_ScannerWriteData.TcDUT (not stored), ST_SickScannerBase.TcDUT (not stored), ST_SickScannerStates.TcDUT (not stored)
//   20_Product/20_ProBox/22_ProMove/11_Addons/91_SickScannerAddon/10_App/ FB_ReadFileLine.TcPOU (not stored), FB_SickScannerAddon.TcPOU (not stored), FB_SickScannerAddonCLV690.TcPOU (not stored), FB_SickScannerBase.TcPOU (not stored)
//   20_Product/20_ProBox/22_ProMove/11_Addons/91_SickScannerAddon/11_Emu/01_DUTs/ ST_CFG_SickScannerEmulation.TcDUT (not stored)
//   20_Product/20_ProBox/22_ProMove/11_Addons/91_SickScannerAddon/11_Emu/ FB_SickScannerAddonEmulation.TcPOU (not stored)
//   20_Product/20_ProBox/22_ProMove/11_Addons/92_TLB4WeightAddon/10_App/DUTs/ E_TLB4WeightState.TcDUT (not stored), ST_CFG_TLB4Weight.TcDUT (not stored), ST_CtrlInTLB4Weight.TcDUT (not stored), ST_HW_InputsTLB4Weight.TcDUT (not stored), ST_HW_OutputsTLB4Weight.TcDUT (not stored), ST_InputsTLB4Weight.TcDUT (not stored), ST_OutputsTLB4Weight.TcDUT (not stored), ST_TLB4WeightStates.TcDUT (not stored), U_HW_OutputCommands.TcDUT (not stored), U_HW_OutPutExchangeRegister.TcDUT (not stored)
//   20_Product/20_ProBox/22_ProMove/11_Addons/92_TLB4WeightAddon/10_App/ FB_TLB4WeightAddon.TcPOU (not stored)
//   20_Product/20_ProBox/22_ProMove/11_Addons/92_TLB4WeightAddon/11_Emu/ FB_TLB4WeightAddonEmulation.TcPOU (not stored)
//   20_Product/20_ProBox/22_ProMove/11_Addons/93_RejectPanelAddon/10_App/01_DUTs/ E_RejectPanelState.TcDUT (not stored), ST_CFG_RejectPanel.TcDUT (not stored), ST_CtrlInRejectPanel.TcDUT (not stored), ST_CtrlOutRejectPanel.TcDUT (not stored), ST_HW_InputsRejectPanel.TcDUT (not stored), ST_HW_OutputsRejectPanel.TcDUT (not stored), ST_InputsRejectPanel.TcDUT (not stored), ST_MaxProfileValues.TcDUT (not stored), ST_OutputsRejectPanel.TcDUT (not stored), ST_RejectPanelStates.TcDUT (not stored)
//   20_Product/20_ProBox/22_ProMove/11_Addons/93_RejectPanelAddon/10_App/ FB_RejectPanelAddon.TcPOU (not stored), F_PalletEvaluation.TcPOU (not stored)
//   20_Product/20_ProBox/22_ProMove/11_Addons/93_RejectPanelAddon/11_Emu/ FB_RejectPanelAddonEmulation.TcPOU (not stored)
//   20_Product/20_ProBox/22_ProMove/11_Addons/94_PalletCheckAddon/10_App/01_DUTs/ E_PalletCheckStates.TcDUT (not stored), ST_CFG_PalletCheck.TcDUT (not stored), ST_CtrlInPalletCheck.TcDUT (not stored), ST_HW_InputsPalletCheck.TcDUT (not stored), ST_InputsPalletCheck.TcDUT (not stored)
//   20_Product/20_ProBox/22_ProMove/11_Addons/94_PalletCheckAddon/10_App/ FB_PalletCheckAddon.TcPOU (not stored)
//   20_Product/20_ProBox/22_ProMove/11_Addons/94_PalletCheckAddon/11_Emu/ FB_PalletCheckAddonEmulation.TcPOU (not stored)
//   20_Product/20_ProBox/22_ProMove/11_Addons/95_RunnerCheckAddon/10_App/01_DUTs/ E_RunnerCheckStates.TcDUT (not stored), ST_CFG_RunnerCheck.TcDUT (not stored), ST_CtrlInRunnerCheck.TcDUT (not stored), ST_CtrlOut_RunnerCheck.TcDUT (not stored), ST_HW_InputsRunnerCheck.TcDUT (not stored), ST_InputsRunnerCheck.TcDUT (not stored), ST_RunnerCheckData.TcDUT (not stored)
//   20_Product/20_ProBox/22_ProMove/11_Addons/95_RunnerCheckAddon/10_App/ FB_RunnerCheckAddon.TcPOU (not stored)
//   20_Product/20_ProBox/22_ProMove/11_Addons/95_RunnerCheckAddon/11_Emu/ FB_RunnerCheckAddonEmulation.TcPOU (not stored)
//   20_Product/20_ProBox/22_ProMove/11_Addons/96_ClosedPalletCheck/10_App/01_DUTs/ E_ClosedPalletCheckStates.TcDUT (not stored), ST_CFG_ClosedPalletCheck.TcDUT (not stored), ST_ClosedPalletCheckStates.TcDUT (not stored), ST_CtrlInClosedPalletCheck.TcDUT (not stored), ST_HW_InputsClosedPalletCheck.TcDUT (not stored), ST_HW_OutputsClosedPalletCheck.TcDUT (not stored), ST_InputsClosedPalletCheck.TcDUT (not stored), ST_OutputsClosedPalletCheck.TcDUT (not stored)
//   20_Product/20_ProBox/22_ProMove/11_Addons/96_ClosedPalletCheck/10_App/ FB_ClosedPalletCheckAddon.TcPOU (not stored)
//   20_Product/20_ProBox/22_ProMove/11_Addons/96_ClosedPalletCheck/11_Emu/ FB_ClosedPalletCheckAddonEmulation.TcPOU (not stored)
//   20_Product/20_ProBox/22_ProMove/11_Addons/ FB_AddOnErrHandler.TcPOU
//   20_Product/20_ProBox/22_ProMove/12_Functions/11_StraightTransport/10_App/01_DUTs/ ST_CFG_ProBoxStraightTransport.TcDUT (not stored), ST_CtrlInPbStraightTransport.TcDUT (not stored), ST_HW_InputsProBoxStraightTransport.TcDUT (not stored), ST_InputsProBoxStraightTransport.TcDUT (not stored)
//   20_Product/20_ProBox/22_ProMove/12_Functions/11_StraightTransport/10_App/01_DUTs_Base/ ST_StraightBase.TcDUT (not stored), ST_StraightBaseZoneOrders.TcDUT (not stored)
//   20_Product/20_ProBox/22_ProMove/12_Functions/11_StraightTransport/10_App/ FB_ProBoxStraightTransport.TcPOU (not stored), FB_StraightBase.TcPOU (not stored)
//   20_Product/20_ProBox/22_ProMove/12_Functions/11_StraightTransport/11_Emu/01_DUTs/ ST_DebugSensors_ProBoxStraightTransportEmulation.TcDUT (not stored)
//   20_Product/20_ProBox/22_ProMove/12_Functions/11_StraightTransport/11_Emu/ FB_ProBoxStraightTransportEmulation.TcPOU (not stored)
//   20_Product/20_ProBox/22_ProMove/12_Functions/20_TransferUnit/10_App/01_DUTs/ E_LiftType.TcDUT (not stored), E_SingleTuMode.TcDUT (not stored), ST_CFG_TransferUnit.TcDUT (not stored), ST_CtrlInPbTransferUnit.TcDUT (not stored), ST_HW_InputsTransferUnit.TcDUT (not stored), ST_HW_OutputsTransferUnit.TcDUT (not stored), ST_InputsTransferUnit.TcDUT (not stored), ST_OutputsTransferUnit.TcDUT (not stored)
//   20_Product/20_ProBox/22_ProMove/12_Functions/20_TransferUnit/10_App/ FB_TransferUnit.TcPOU (not stored)
//   20_Product/20_ProBox/22_ProMove/12_Functions/20_TransferUnit/11_Emu/01_DUTs/ ST_CFG_TransferUnitEmulation.TcDUT (not stored), ST_DebugSensors_TransferUnitEmulation.TcDUT (not stored)
//   20_Product/20_ProBox/22_ProMove/12_Functions/20_TransferUnit/11_Emu/ FB_TransferUnitEmulation.TcPOU (not stored)
//   20_Product/20_ProBox/22_ProMove/12_Functions/21_LowLiftUnit/10_App/01_DUTs/ ST_CFG_LowLiftUnit.TcDUT (not stored), ST_HW_InputsLowLiftUnit.TcDUT (not stored), ST_HW_OutputsLowLiftUnit.TcDUT (not stored), ST_InputsLowLiftUnit.TcDUT (not stored), ST_OutputsLowLiftUnit.TcDUT (not stored)
//   20_Product/20_ProBox/22_ProMove/12_Functions/21_LowLiftUnit/10_App/ FB_LowLiftUnit.TcPOU (not stored)
//   20_Product/20_ProBox/22_ProMove/12_Functions/21_LowLiftUnit/11_Emu/01_DUTs/ ST_CFG_LowLiftUnitEmulation.TcDUT (not stored), ST_DebugSensors_LowLiftEmulation.TcDUT (not stored)
//   20_Product/20_ProBox/22_ProMove/12_Functions/21_LowLiftUnit/11_Emu/ FB_LowLiftUnitEmulation.TcPOU (not stored)
//   20_Product/20_ProBox/22_ProMove/12_Functions/22_TurnTable/10_App/01_DUTs_Base/ E_AdjacentSideType.TcDUT (not stored), ST_CtrlInTT.TcDUT (not stored), ST_HW_InputsTT.TcDUT (not stored), ST_HW_InputsTTConv.TcDUT (not stored), ST_TTDriveReq.TcDUT (not stored)
//   20_Product/20_ProBox/22_ProMove/12_Functions/22_TurnTable/10_App/01_DUTs_TurnTableDTU/ ST_CFG_TurnTableDTU.TcDUT (not stored), ST_HW_InputsTurnTableDTU.TcDUT (not stored), ST_HW_OutputsTurnTableDTU.TcDUT (not stored)
//   20_Product/20_ProBox/22_ProMove/12_Functions/22_TurnTable/10_App/01_DUTs_TurnTable/ ST_CFG_TurnTable.TcDUT (not stored), ST_HW_InputsTurnTable.TcDUT (not stored), ST_HW_OutputsTurnTable.TcDUT (not stored)
//   20_Product/20_ProBox/22_ProMove/12_Functions/22_TurnTable/10_App/ FB_TurnTable.TcPOU (not stored), FB_TurnTableBase.TcPOU (not stored), FB_TurnTableDtu.TcPOU (not stored)
//   20_Product/20_ProBox/22_ProMove/12_Functions/22_TurnTable/11_Emu/01_DUTs/ ST_CFG_TurnTableDtuEmulation.TcDUT (not stored), ST_CFG_TurnTableEmulation.TcDUT (not stored), ST_CFG_TurnTablePositionEmu.TcDUT (not stored), ST_DebugSensors_TurnTableDtuEmulation.TcDUT (not stored), ST_DebugSensors_TurnTableEmulation.TcDUT (not stored)
//   20_Product/20_ProBox/22_ProMove/12_Functions/22_TurnTable/11_Emu/ FB_TurnTableDtuEmulation.TcPOU (not stored), FB_TurnTableEmulation.TcPOU (not stored)
//   20_Product/20_ProBox/22_ProMove/12_Functions/28_TransferCC/10_App/01_DUTs/ ST_CFG_TransferCC.TcDUT (not stored), ST_HW_InputsTransferCC.TcDUT (not stored), ST_HW_OutputsTransferCC.TcDUT (not stored), ST_InputsTransferCC.TcDUT (not stored), ST_OutputsTransferCC.TcDUT (not stored)
//   20_Product/20_ProBox/22_ProMove/12_Functions/28_TransferCC/10_App/ FB_TransferCC.TcPOU (not stored)
//   20_Product/20_ProBox/22_ProMove/12_Functions/28_TransferCC/11_Emu/01_DUTs/ ST_CFG_TransferCCEmulation.TcDUT (not stored), ST_DebugSensors_TransferCCEmulation.TcDUT (not stored)
//   20_Product/20_ProBox/22_ProMove/12_Functions/28_TransferCC/11_Emu/ FB_TransferCC_Emulation.TcPOU (not stored)
//   20_Product/20_ProBox/22_ProMove/12_Functions/29_Sideshift/10_App/01_DUTs/ ST_CFG_Sideshift.TcDUT (not stored), ST_HW_InputsSideshift.TcDUT (not stored), ST_HW_OutputsSideshift.TcDUT (not stored), ST_InputsSideshift.TcDUT (not stored), ST_OutputsSideshift.TcDUT (not stored)
//   20_Product/20_ProBox/22_ProMove/12_Functions/29_Sideshift/10_App/ FB_Sideshift.TcPOU (not stored)
//   20_Product/20_ProBox/22_ProMove/12_Functions/29_Sideshift/11_Emu/01_DUTs/ ST_CFG_SideShiftEmulation.TcDUT (not stored), ST_DebugSensors_SideshiftEmulation.TcDUT (not stored)
//   20_Product/20_ProBox/22_ProMove/12_Functions/29_Sideshift/11_Emu/ FB_Sideshift_Emulation.TcPOU (not stored)
//   20_Product/20_ProBox/22_ProMove/12_Functions/80_FunctionForks/10_App/01_DUTs/ E_FunctionForkOrder.TcDUT (not stored), E_FunctionForkState.TcDUT (not stored), ST_CFG_FunctionForks.TcDUT (not stored), ST_CtrlOutFunctionForks.TcDUT (not stored), ST_ForkRequest.TcDUT (not stored), ST_ForkState.TcDUT (not stored), ST_FunctionForkData.TcDUT (not stored), ST_FunctionForkManualCtrl.TcDUT (not stored), ST_HW_InputsFunctionFork.TcDUT (not stored), ST_HW_OutputsFunctionForks.TcDUT (not stored), ST_InputsFunctionForks.TcDUT (not stored), ST_OutputsFunctionForks.TcDUT (not stored)
//   20_Product/20_ProBox/22_ProMove/12_Functions/80_FunctionForks/10_App/ FB_ElementForkInterface.TcPOU (not stored), FB_FunctionForks.TcPOU (not stored), ITF_PB_ElementForkInterface.TcIO (not stored)
//   20_Product/20_ProBox/22_ProMove/12_Functions/80_FunctionForks/11_Emu/ FB_FunctionForksEmulation.TcPOU (not stored)
//   20_Product/20_ProBox/22_ProMove/13_Elements/11_ElementMotor/10_App/01_DUTs/ ST_CFG_ProBoxElementBase.TcDUT (not stored), ST_CFG_ProBoxElementMotor.TcDUT (not stored), ST_ElementSpeed.TcDUT (not stored), ST_HW_InputsProBoxElementMotor.TcDUT (not stored), ST_HW_OutputsProBoxElementMotor.TcDUT (not stored), ST_InputsProBoxElementMotor.TcDUT (not stored)
//   20_Product/20_ProBox/22_ProMove/13_Elements/11_ElementMotor/10_App/ FB_PB_Element_Encoder.TcPOU (not stored), FB_ProBoxElementBase.TcPOU (not stored), FB_ProBoxElementMotor.TcPOU (not stored), ITF_PB_Element.TcIO (not stored)
//   20_Product/20_ProBox/22_ProMove/13_Elements/11_ElementMotor/11_Emu/ FB_ProBoxElementMotorEmulation.TcPOU (not stored)
//   20_Product/20_ProBox/22_ProMove/13_Elements/12_Element2Motor/10_App/01_DUTs/ ST_HW_OutputsProBoxElement2Motor.TcDUT (not stored)
//   20_Product/20_ProBox/22_ProMove/13_Elements/12_Element2Motor/10_App/ FB_ProBoxElement2Motor.TcPOU (not stored)
//   20_Product/20_ProBox/22_ProMove/13_Elements/12_Element2Motor/11_Emu/ FB_ProBoxElement2MotorEmulation.TcPOU (not stored)
//   20_Product/20_ProBox/22_ProMove/13_Elements/14_ElementMPD/10_App/01_DUTs_Base/ ST_HW_OutputsMotionDrive.TcDUT (not stored), ST_MPD_ExternalErrors.TcDUT (not stored)
//   20_Product/20_ProBox/22_ProMove/13_Elements/14_ElementMPD/10_App/01_DUTs_ShuttleForks/ ST_CFG_PDs_ShuttleForks.TcDUT (not stored), ST_CFG_ProBoxElementShuttleForks.TcDUT (not stored), ST_CFG_ShuttleForkLift.TcDUT (not stored), ST_HW_InputsProBoxElementShuttleForks.TcDUT (not stored), ST_HW_Inputs_Conv_ShuttleForks.TcDUT (not stored), ST_HW_OutputsProBoxElementShuttleForks.TcDUT (not stored), ST_ShuttleForkData.TcDUT (not stored), ST_ShuttleForkLift.TcDUT (not stored), ST_ShuttleLiftData.TcDUT (not stored)
//   20_Product/20_ProBox/22_ProMove/13_Elements/14_ElementMPD/10_App/01_DUTs_Shuttle/ E_CFG_Tilt.TcDUT (not stored), ST_CFG_PDs_Shuttle.TcDUT (not stored), ST_CFG_ProBoxElementShuttle.TcDUT (not stored), ST_HW_InputsMPD_Conv_Shuttle.TcDUT (not stored), ST_HW_InputsProBoxElementShuttle.TcDUT (not stored), ST_HW_OutputsProBoxElementMotorShuttle.TcDUT (not stored), ST_HW_OutputsProBoxElementShuttle.TcDUT (not stored)
//   20_Product/20_ProBox/22_ProMove/13_Elements/14_ElementMPD/10_App/01_DUTs_VC/ ST_CFG_ProBoxElementVC.TcDUT (not stored), ST_CFG_ProBoxElementVcBase.TcDUT (not stored), ST_HW_InputsProBoxElementVC.TcDUT (not stored), ST_HW_OutputsElementVC_Base.TcDUT (not stored), ST_HW_OutputsProBoxElementVC.TcDUT (not stored), ST_VC_CFG_PDs.TcDUT (not stored), ST_VC_ForkData.TcDUT (not stored)
//   20_Product/20_ProBox/22_ProMove/13_Elements/14_ElementMPD/10_App/ FB_ElementMpdBase.TcPOU (not stored), FB_ProBoxElementShuttle.TcPOU (not stored), FB_ProBoxElementShuttleForks.TcPOU (not stored), FB_ProBoxElementVC.TcPOU (not stored), FB_ProBoxElementVC_Base.TcPOU (not stored)
//   20_Product/20_ProBox/22_ProMove/13_Elements/14_ElementMPD/11_Emu/ FB_ProBoxElementShuttleEmulation.TcPOU (not stored), FB_ProBoxElementShuttleForksEmulation.TcPOU (not stored), FB_ProBoxElementVC_Emulation.TcPOU (not stored), F_MPD_GetOverhangSensorStatus.TcPOU (not stored)
//   20_Product/20_ProBox/22_ProMove/14_Groups/10_App/00_GVLs/ GVL_PB_SG.TcGVL (not stored)
//   20_Product/20_ProBox/22_ProMove/14_Groups/10_App/01_DUTs/Cabinet/ ST_PB_SG_Cabinet.TcDUT (not stored), ST_PB_SG_CabinetInputExt.TcDUT (not stored), ST_PB_SG_DiagInputs.TcDUT (not stored)
//   20_Product/20_ProBox/22_ProMove/14_Groups/10_App/01_DUTs/ ST_CFG_ProBoxSG.TcDUT (not stored), ST_CtlrOutProBoxSG.TcDUT (not stored), ST_EmgStatus.TcDUT (not stored), ST_HW_InputsSG_ProBOX.TcDUT (not stored), ST_HW_OutputsSG_ProBOX.TcDUT (not stored), ST_PB_SG_InputsCommand.TcDUT (not stored), ST_SG_InputsSignals_ProBOX.TcDUT (not stored), ST_SG_Inputs_ProBOX.TcDUT (not stored), ST_SG_Outputs_ProBOX.TcDUT (not stored)
//   20_Product/20_ProBox/22_ProMove/14_Groups/10_App/ FB_ProBOXSG.TcPOU, F_DebugUseEmuVizu.TcPOU
//   20_Product/20_ProBox/22_ProMove/14_Groups/11_Emu/01_DUTs/ ST_CFG_ProBoxSGEmulation.TcDUT (not stored)
//   20_Product/20_ProBox/22_ProMove/14_Groups/11_Emu/ FB_ProBOXSG_Emulation.TcPOU
//   20_Product/20_ProBox/22_ProMove/15_SubSystem/01_DUTs/ ST_CFG_ProBoxSubsystem.TcDUT
//   20_Product/20_ProBox/22_ProMove/15_SubSystem/ FB_ProBoxSubsystem.TcPOU, FB_ProBoxSubsystemEmulation.TcPOU
//   20_Product/20_ProBox/30_Toolbox/11_Emu/ F_AddPhysicalTU.TcPOU, F_RemovePhysicalTU.TcPOU
//   20_Product/20_ProBox/30_Toolbox/12_DUTs/ E_PalletOrientation.TcDUT
//   20_Product/20_ProBox/30_Toolbox/70_Strategies/01_DUTs/ GVL_Strategies.TcGVL, ST_FifoBuffer.TcDUT, ST_RoutingSluggingData.TcDUT
//   20_Product/20_ProBox/30_Toolbox/70_Strategies/ FB_CountTUs.TcPOU, FB_DTU_MergingControl.TcPOU, FB_LoopControl.TcPOU, FB_MergingFiFo.TcPOU, F_PB_RoutingSlugging.TcPOU
//   20_Product/20_ProBox/30_Toolbox/71_SafetyInterface/01_AK_Cabinet/01_DUTs/ ST_ProBoxSafetyAK.TcDUT (not stored), ST_ProBoxSafetyInputsAK.TcDUT (not stored), ST_ProBoxSafetyOutputsAK.TcDUT (not stored)
//   20_Product/20_ProBox/30_Toolbox/71_SafetyInterface/01_AK_Cabinet/ FB_SafetySignalsAK.TcPOU
//   20_Product/20_ProBox/30_Toolbox/71_SafetyInterface/02_LowLift/01_DUTs/ ST_ProBoxSafetyInputsLowLift.TcDUT (not stored), ST_ProBoxSafetyLowLift.TcDUT (not stored), ST_ProBoxSafetyOutputsLowLift.TcDUT (not stored)
//   20_Product/20_ProBox/30_Toolbox/71_SafetyInterface/02_LowLift/ FB_SafetySignalsLowLift.TcPOU
//   20_Product/20_ProBox/30_Toolbox/71_SafetyInterface/03_Shuttle/01_DUTs/ ST_ProBoxSafetyInputsShuttle.TcDUT (not stored), ST_ProBoxSafetyOutputsShuttle.TcDUT (not stored), ST_ProBoxSafetyShuttle.TcDUT (not stored)
//   20_Product/20_ProBox/30_Toolbox/71_SafetyInterface/03_Shuttle/ FB_SafetySignalsShuttle.TcPOU
//   20_Product/20_ProBox/30_Toolbox/71_SafetyInterface/04_VerticalConveyor/01_DUTs/ ST_ProBoxSafetyInputsVerticalConv.TcDUT (not stored), ST_ProBoxSafetyOutputsVerticalConv.TcDUT (not stored), ST_ProBoxSafetyVerticalConv.TcDUT (not stored)
//   20_Product/20_ProBox/30_Toolbox/71_SafetyInterface/04_VerticalConveyor/ FB_SafetySignalsVerticalConv.TcPOU
//   20_Product/20_ProBox/30_Toolbox/71_SafetyInterface/SafetyZoneSignals/01_DUTs/ ST_ProBoxSafetyInputsSZPCo.TcDUT (not stored), ST_ProBoxSafetyOutputsSZPCo.TcDUT (not stored), ST_ProBoxSafetySZPCo.TcDUT (not stored)
//   20_Product/20_ProBox/30_Toolbox/71_SafetyInterface/SafetyZoneSignals/ FB_SafetySignalsSZPCo.TcPOU
//   20_Product/20_ProBox/30_Toolbox/ FB_ClockHz.TcPOU, FB_CountTUDestination.TcPOU, FB_FunctionOrdersToProBox.TcPOU, FB_PAC_CapacityCounter.TcPOU, FB_PB_PresetEncoder.TcPOU, FB_SendTelegram.TcPOU, F_AssignTU_DataIndexToZone.TcPOU, F_CheckAllEnabled.TcPOU, F_CheckAllFree.TcPOU, F_CheckAllOccupied.TcPOU, F_CheckAllStarted.TcPOU, F_DeleteTU_DataIndex.TcPOU, F_PB_GetAdjacentFunctionZoneIndex.TcPOU, F_PB_GetTransportControlDataRef.TcPOU, F_PB_GetTransportData.TcPOU, F_PB_GetTuDestination.TcPOU, F_PB_GetZoneITC.TcPOU, F_PB_IsLogicalOccupied.TcPOU, F_PB_SetDestination.TcPOU, F_PB_SetPalletOrientation.TcPOU, F_ResetOccupied.TcPOU, F_SetOccupied.TcPOU
//   20_Product/20_ProBox/40_TC_Visualization/10_Controls/LoopControl/ V_LoopControl.TcVIS
//   20_Product/20_ProBox/40_TC_Visualization/10_Controls/TransportControl/ V_TransportControl.TcVIS
//   20_Product/20_ProBox/40_TC_Visualization/11_Addon/CraneXoverAddon/ V_CraneXoverAddon.TcVIS
//   20_Product/20_ProBox/40_TC_Visualization/11_Addon/FastDoorAddon/ V_FastDoorAddon.TcVIS
//   20_Product/20_ProBox/40_TC_Visualization/11_Addon/InOutFeedAddon/ V_InOutFeedAddon.TcVIS
//   20_Product/20_ProBox/40_TC_Visualization/11_Addon/LiftTableAddon/ V_LiftTableAddon.TcVIS
//   20_Product/20_ProBox/40_TC_Visualization/11_Addon/PalletCheckAddon/ V_PalletCheckAddon.TcVIS
//   20_Product/20_ProBox/40_TC_Visualization/11_Addon/PalletMagazineAddon/ V_PalletMagazineAddon.TcVIS
//   20_Product/20_ProBox/40_TC_Visualization/11_Addon/ProfileCheckAddon/ V_ProfileCheckAddon.TcVIS
//   20_Product/20_ProBox/40_TC_Visualization/11_Addon/RejectPanelAddon/ V_RejectPanelAddon.TcVIS
//   20_Product/20_ProBox/40_TC_Visualization/11_Addon/SickScannerAddon/ V_SickScannerAddon.TcVIS
//   20_Product/20_ProBox/40_TC_Visualization/11_Addon/TLB4WeightAddon/ V_TLB4WeightAddon.TcVIS
//   20_Product/20_ProBox/40_TC_Visualization/12_Functions/FunctionForks/ V_FunctionFork.TcVIS
//   20_Product/20_ProBox/40_TC_Visualization/12_Functions/LowLiftUnit/ V_LowLiftUnit.TcVIS
//   20_Product/20_ProBox/40_TC_Visualization/12_Functions/ProBoxStraightTransport/ V_ProBoxStraightTransport.TcVIS
//   20_Product/20_ProBox/40_TC_Visualization/12_Functions/TransferCC/ V_TransferCC.TcVIS
//   20_Product/20_ProBox/40_TC_Visualization/12_Functions/TransferUnit/ V_TransferUnit.TcVIS
//   20_Product/20_ProBox/40_TC_Visualization/12_Functions/TurnTable/ V_TurnTable.TcVIS
//   20_Product/20_ProBox/40_TC_Visualization/13_Elements/ V_Element_Shuttle.TcVIS, V_Element_VC.TcVIS
//   20_Product/20_ProBox/40_TC_Visualization/14_Group/ V_Group.TcVIS
//   20_Product/20_ProBox/40_TC_Visualization/15_PowerStore/ AccessPanelCmbTxtList.TcTLO, AkCmbTxtList.TcTLO, LevelCmbTxtList.TcTLO, PanelCmbTxtList.TcTLO, SymbolPool.TcIPO (not stored), TransferPanelCmbTxtList.TcTLO, V_AccessPanel.TcVIS, V_AKcabinetPanel.TcVIS, V_AkPanelSelecCmb.TcVIS, V_ApSelecCmb.TcVIS, V_LevelSelecCmb.TcVIS, V_PanelSelecCmb.TcVIS, V_TpSelecCmb.TcVIS, V_TransferPanel.TcVIS, V_VC_AccessPanel.TcVIS
//   20_Product/20_ProBox/40_TC_Visualization/15_PowerStore/DTUs/ ST_AccessPanel.TcDUT, ST_AccessPanelInputs.TcDUT, ST_AccessPanelOutputs.TcDUT, ST_AKcabinetPanel.TcDUT, ST_AKcabinetPanelInputs.TcDUT, ST_AKcabinetPanelOutputs.TcDUT, ST_TransferPanel.TcDUT, ST_TransferPanelInputs.TcDUT, ST_TransferPanelOutputs.TcDUT, ST_VC_AccessPanel.TcDUT, ST_VC_AccessPanelInputs.TcDUT, ST_VC_AccessPanelOutputs.TcDUT
//   20_Product/20_ProBox/40_TC_Visualization/99_SIS/ FB_VizuSIS.TcPOU, V_SIS_Control.TcVIS
//   20_Product/20_ProBox/ MainProBox.TcPOU, ProBox_Version.TcTLO
//   20_Product/30_Toolbox/11_Com/10_TCP_Driver/01_DUTs/ E_ConnStates.TcDUT, E_RecvStates.TcDUT, E_SendStates.TcDUT, E_ServStates.TcDUT, ST_CFG_TcpDriver.TcDUT
//   20_Product/30_Toolbox/11_Com/10_TCP_Driver/ FB_TCP_Driver.TcPOU
//   20_Product/30_Toolbox/12_StringStream/ F_AssembleByteStream.TcPOU, F_CompareAlphaNumericString.TcPOU, F_MaxReportTime_TO_Time.TcPOU, F_ReduceToAlphaNumeric.TcPOU, F_RemoveSign.TcPOU, F_SampleTime_TO_TIME.TcPOU, F_StuffString.TcPOU, F_Time_TO_MaxReportTime.TcPOU, F_Time_TO_SampleTime.TcPOU
//   20_Product/30_Toolbox/13_TimerCounter/01_DUTs/ E_PulsGen.TcDUT
//   20_Product/30_Toolbox/13_TimerCounter/ FB_GeneratePulse.TcPOU, FB_Timer.TcPOU
//   20_Product/30_Toolbox/16_Sequencing/00_GVLs/ SequencingParameter.TcGVL
//   20_Product/30_Toolbox/16_Sequencing/01_DUTs/ ST_SeqEntry.TcDUT
//   20_Product/30_Toolbox/16_Sequencing/02_ITFs/ I_BranchCheckpoint.TcIO, I_SeqEstimateNext.TcIO
//   20_Product/30_Toolbox/16_Sequencing/10_Core/ FB_SeqBranch.TcPOU, FB_SeqBranchMux.TcPOU, FB_SeqBuildStream.TcPOU, FB_SeqGetNextTU.TcPOU, FB_SeqLimitedStream.TcPOU, FB_SeqReleaseRequest.TcPOU, F_UpdateCheckpointID.TcPOU
//   20_Product/30_Toolbox/16_Sequencing/11_Strategies/ FB_SeqCheckpoint.TcPOU, FB_SeqEstimateAllNextTUs.TcPOU, FB_SeqEstimateNextTU.TcPOU, FB_SeqEstimateStreamRange.TcPOU, FB_SeqMerge2W.TcPOU
//   20_Product/30_Toolbox/16_Sequencing/12_Helper/ FB_SeqConveyorLane.TcPOU
//   20_Product/30_Toolbox/17_WindowTracking/10_Core/00_GVLs/ WindowTracking.TcGVL
//   20_Product/30_Toolbox/17_WindowTracking/10_Core/01_DUTs/ E_WindowTrackingWindowState.TcDUT, ST_WindowTrackingReloc.TcDUT, ST_WindowTrackingTransfer.TcDUT, ST_WindowTrackingWindow.TcDUT, ST_WindowTrackingZone.TcDUT, ST_ZoneDataPair.TcDUT
//   20_Product/30_Toolbox/17_WindowTracking/10_Core/02_ITFs/ I_Encoder.TcIO, I_TrackingActionListener.TcIO, I_TrackingMaster.TcIO, I_WindowTracking.TcIO, I_WindowTrackingListener.TcIO
//   20_Product/30_Toolbox/17_WindowTracking/10_Core/ FB_DisplacementMeter.TcPOU, FB_EncoderEx.TcPOU, FB_WindowRelocator.TcPOU, FB_WindowTracking.TcPOU
//   20_Product/30_Toolbox/99_Misc/01_DUTs/ E_CPU_InfoStates.TcDUT
//   20_Product/30_Toolbox/99_Misc/13_Helper/01_DUTs/ ST_TrackingZoneInfo.TcDUT
//   20_Product/30_Toolbox/99_Misc/13_Helper/ FB_EncoderMonitor.TcPOU, FB_FindTrackingZones.TcPOU, FB_MeasureEncoderResolution.TcPOU, FB_ScaleEncoder.TcPOU, FB_Throughput.TcPOU, FB_TrackingReservation.TcPOU, F_AlignEncoderValue.TcPOU, F_CountTUs.TcPOU, F_CountTUsWithDestination.TcPOU
//   20_Product/30_Toolbox/99_Misc/ FB_Encoder.TcPOU, FB_SystemInfo.TcPOU, F_BlockCopy.TcPOU, F_CreateHashCode.TcPOU
//   / PlcTask.TcTTO, Visualization Manager.TcVMO (not stored)

CONFIGURATION PLC_1
    RESOURCE PLC ON TwinCAT3
        TASK PlcTask(INTERVAL := T#10ms, PRIORITY := 20);
        PROGRAM MainProBox WITH PlcTask : MainProBox;
    END_RESOURCE
END_CONFIGURATION

// ---- 10_Project/10_App/10_Config/01_DUTs/E_ElementNumber.TcDUT
///Automatically generated by BoxConfigurator 
TYPE E_ElementNumber :
(
	E_BEGIN_ELEMENT,
	E_10_001_0200_00_0,
	E_10_001_0201_00_0,
	E_10_001_0202_00_0,
	E_10_001_0203_00_0,
	E_10_001_0204_00_0,
	E_10_001_0205_00_0,
	E_10_001_0207_00_0,
	E_10_001_0208_00_0,
	E_10_001_0209_00_0,
	E_10_001_0211_00_0,
	E_10_001_0212_00_0,
	E_10_001_0213_00_0,
	E_10_001_0214_00_0,
	E_10_001_0215_00_0,
	E_10_001_0216_00_0,
	E_10_001_0217_00_0,
	E_10_001_0218_00_0,
	E_10_001_0219_00_0,
	E_10_001_0220_00_0,
	E_10_001_0221_00_0,
	E_10_001_0222_00_0,
	E_10_001_0223_00_0,
	E_10_001_0225_00_0,
	E_10_001_0226_00_0,
	E_10_001_0227_00_0,
	E_10_001_0230_00_0,
	E_10_001_0232_00_0,
	E_10_001_0233_00_0,
	E_10_002_0206_00_0,
	E_END_ELEMENT
);
END_TYPE

// ---- 10_Project/10_App/10_Config/01_DUTs/E_FunctionNumber.TcDUT
///Automatically generated by BoxConfigurator 
TYPE E_FunctionNumber :
(
	F_BEGIN_FUNCTION,
	F_10_001_0200_01_0,
	F_10_001_0200_02_0,
	F_10_001_0201_01_0,
	F_10_001_0202_01_0,
	F_10_001_0203_01_0,
	F_10_001_0203_02_0,
	F_10_001_0203_03_0,
	F_10_001_0203_04_0,
	F_10_001_0203_05_0,
	F_10_001_0204_01_0,
	F_10_001_0207_01_0,
	F_10_001_0207_02_0,
	F_10_001_0208_01_0,
	F_10_001_0209_01_0,
	F_10_001_0211_01_0,
	F_10_001_0212_01_0,
	F_10_001_0213_01_0,
	F_10_001_0213_02_0,
	F_10_001_0214_01_0,
	F_10_001_0215_01_0,
	F_10_001_0215_02_0,
	F_10_001_0215_03_0,
	F_10_001_0216_01_0,
	F_10_001_0216_02_0,
	F_10_001_0217_01_0,
	F_10_001_0218_01_0,
	F_10_001_0219_01_0,
	F_10_001_0220_01_0,
	F_10_001_0221_01_0,
	F_10_001_0222_01_0,
	F_10_001_0225_01_0,
	F_10_001_0226_01_0,
	F_10_001_0227_01_0,
	F_10_001_0230_01_0,
	F_10_001_0232_01_0,
	F_10_001_0232_02_0,
	F_10_001_0233_01_0,
	F_10_002_0206_01_0,
	F_END_FUNCTION,
	F_BEGIN_EXTERN_FUNCTION,
	F_END_EXTERN_FUNCTION,
	F_BEGIN_VIRTUAL_FUNCTION,
	F_END_VIRTUAL_FUNCTION
);
END_TYPE

// ---- 10_Project/10_App/10_Config/01_DUTs/E_GroupNumber.TcDUT
///Automatically generated by BoxConfigurator 
TYPE E_GroupNumber :
(
	G_BEGIN_GROUP,
	G_SG_001,
	G_SG_002,
	G_END_GROUP
);
END_TYPE

// ---- 20_Product/10_BCF/10_Base/01_DUTs/E_CM_Index.TcDUT
TYPE E_CM_Index :
(**************************************************************************************
 * 	Application		:	BoxControl Framework
 *	Revision		:	$Revision: 404529 $
 *	Revision date	:	$Date: 2018-04-23 08:21:38 +0200 (Mo., 23 Apr 2018) $
 *	Last changed by	:	$Author: b7bolm $
 *	URL				:	$URL: http://almscdc.swisslog.com/repo/SWPD/Development/BoxControlFramework/20_Release/trunk/01_Software/BCF/BCF/JumpStart/20_Product/10_App/10_Base/10_Lib/01_DUTs/E_CM_Index.TcDUT $
 *
 *	Purpose			:	Index for condition Monitoring Variable Storage					
 *
 *
 * ------------------------------------------------------------------------------------
 *	Copyright Swisslog [IP AG], Switzerland. All rights reserved.
 * 
 * ------------------------------------------------------------------------------------
 *	
 * 	Revision History: 
 *
 * 	VERSION			DATE			INITIALS			DESCRIPTION
 *	0.1				01.01.2001		swl					Example
 *
 **************************************************************************************)	
(
	E_BEGIN_VARIABLE,
	CM01, 
	CM02,
	CM03,
	CM04,
	CM05,
	CM06,
	E_END_VARIABLE
);
END_TYPE

// ---- 20_Product/10_BCF/10_Base/01_DUTs/E_CM_Mode.TcDUT
TYPE E_CM_Mode :
(**************************************************************************************
 * 	Application		:	BoxControl Framework
 *	Revision		:	$Revision: 404529 $
 *	Revision date	:	$Date: 2018-04-23 08:21:38 +0200 (Mo., 23 Apr 2018) $
 *	Last changed by	:	$Author: b7bolm $
 *	URL				:	$URL: http://almscdc.swisslog.com/repo/SWPD/Development/BoxControlFramework/20_Release/trunk/01_Software/BCF/BCF/JumpStart/20_Product/10_App/10_Base/10_Lib/01_DUTs/E_CM_Mode.TcDUT $
 *
 *	Purpose			:	Condition Monitoring Mode Enumeration  					
 *
 *
 * ------------------------------------------------------------------------------------
 *	Copyright Swisslog [IP AG], Switzerland. All rights reserved.
 * 
 * ------------------------------------------------------------------------------------
 *	
 * 	Revision History: 
 *
 * 	VERSION			DATE			INITIALS			DESCRIPTION
 *	0.1				01.01.2001		swl					Example
 *
 **************************************************************************************)	
(
	E_BEGIN_MODE,
	DEFAULT,
	ALPHANUMERIC,
	E_END_MODE
);
END_TYPE

// ---- 20_Product/10_BCF/10_Base/01_DUTs/E_ErrorState.TcDUT
TYPE E_ErrorState :
(**************************************************************************************
 * 	Application		:	BoxControl Framework
 *	Revision		:	$Revision: 404529 $
 *	Revision date	:	$Date: 2018-04-23 08:21:38 +0200 (Mo., 23 Apr 2018) $
 *	Last changed by	:	$Author: b7bolm $
 *	URL				:	$URL: http://almscdc.swisslog.com/repo/SWPD/Development/BoxControlFramework/20_Release/trunk/01_Software/BCF/BCF/JumpStart/20_Product/10_App/10_Base/10_Lib/01_DUTs/E_ErrorState.TcDUT $
 *
 *	Purpose			:	Error states - Order is important
 *
 * ------------------------------------------------------------------------------------
 *	Copyright Swisslog [IP AG], Switzerland. All rights reserved.
 * 
 * ------------------------------------------------------------------------------------
 *	
 * 	Revision History: 
 *
 * 	VERSION			DATE			INITIALS			DESCRIPTION
 *	0.1				01.01.2001		swl					Example
 *
 **************************************************************************************)
(
	UNKNOWN,
	OPERATIONAL,
	WARNING,
	ERROR
);
END_TYPE

// ---- 20_Product/10_BCF/10_Base/01_DUTs/E_ErrorType.TcDUT
TYPE E_ErrorType :
(**************************************************************************************
 * 	Application		:	BoxControl Framework
 *	Revision		:	$Revision: 404529 $
 *	Revision date	:	$Date: 2018-04-23 08:21:38 +0200 (Mo., 23 Apr 2018) $
 *	Last changed by	:	$Author: b7bolm $
 *	URL				:	$URL: http://almscdc.swisslog.com/repo/SWPD/Development/BoxControlFramework/20_Release/trunk/01_Software/BCF/BCF/JumpStart/20_Product/10_App/10_Base/10_Lib/01_DUTs/E_ErrorType.TcDUT $
 *
 *	Purpose			:	Error type
 *
 * ------------------------------------------------------------------------------------
 *	Copyright Swisslog [IP AG], Switzerland. All rights reserved.
 * 
 * ------------------------------------------------------------------------------------
 *	
 * 	Revision History: 
 *
 * 	VERSION			DATE			INITIALS			DESCRIPTION
 *	0.1				01.01.2001		swl					Example
 *
 **************************************************************************************)
(
	NO_ERROR_PENDING,
	INFO,
 	WARNING,
 	ERROR
);
END_TYPE

// ---- 20_Product/10_BCF/10_Base/01_DUTs/E_MFCS_Channel.TcDUT
TYPE E_MFCS_Channel :
(
	BEGIN_CHANNEL,
	AM,
	SPOC,
	LOGGING,
	CM,
	CHANNEL_1,
	CHANNEL_2,
	CHANNEL_3,
	CHANNEL_4,
	CHANNEL_5,
	CHANNEL_6,
	CHANNEL_7,
	END_CHANNEL
);
END_TYPE

// ---- 20_Product/10_BCF/10_Base/01_DUTs/E_PositionMode.TcDUT
TYPE E_PositionMode :
(**************************************************************************************
 * 	Application		:	BoxControl Framework
 *	Revision		:	$Revision: 404529 $
 *	Revision date	:	$Date: 2018-04-23 08:21:38 +0200 (Mo., 23 Apr 2018) $
 *	Last changed by	:	$Author: b7bolm $
 *	URL				:	$URL: http://almscdc.swisslog.com/repo/SWPD/Development/BoxControlFramework/20_Release/trunk/01_Software/BCF/BCF/JumpStart/20_Product/10_App/10_Base/10_Lib/01_DUTs/E_PositionMode.TcDUT $
 *
 *	Purpose			:	Position mode
 *
 * ------------------------------------------------------------------------------------
 *	Copyright Swisslog [IP AG], Switzerland. All rights reserved.
 * 
 * ------------------------------------------------------------------------------------
 *	
 * 	Revision History: 
 *
 * 	VERSION			DATE			INITIALS			DESCRIPTION
 *	0.1				01.01.2001		swl					Example
 *
 **************************************************************************************)
(
	UNKNOWN_MODE,
	OFF_MODE,
	MANUAL_MODE,
	AUTO_MODE,
	SEMI_AUTO
);
END_TYPE

// ---- 20_Product/10_BCF/10_Base/01_DUTs/E_PositionState.TcDUT
TYPE E_PositionState :
(**************************************************************************************
 * 	Application		:	BoxControl Framework
 *	Revision		:	$Revision: 404529 $
 *	Revision date	:	$Date: 2018-04-23 08:21:38 +0200 (Mo., 23 Apr 2018) $
 *	Last changed by	:	$Author: b7bolm $
 *	URL				:	$URL: http://almscdc.swisslog.com/repo/SWPD/Development/BoxControlFramework/20_Release/trunk/01_Software/BCF/BCF/JumpStart/20_Product/10_App/10_Base/10_Lib/01_DUTs/E_PositionState.TcDUT $
 *
 *	Purpose			:	Position states
 *
 * ------------------------------------------------------------------------------------
 *	Copyright Swisslog [IP AG], Switzerland. All rights reserved.
 * 
 * ------------------------------------------------------------------------------------
 *	
 * 	Revision History: 
 *
 * 	VERSION			DATE			INITIALS			DESCRIPTION
 *	0.1				01.01.2001		swl					Example
 *
 **************************************************************************************)
(
	UNKNOWN,
	STOPPED,
	STARTING,
	STOPPING,
	STARTED
);
END_TYPE

// ---- 20_Product/10_BCF/10_Base/01_DUTs/ST_Base.TcDUT
TYPE ST_Base :
(**************************************************************************************
 * 	Application		:	BoxControl Framework
 *	Revision		:	$Revision: 404529 $
 *	Revision date	:	$Date: 2018-04-23 08:21:38 +0200 (Mo., 23 Apr 2018) $
 *	Last changed by	:	$Author: b7bolm $
 *	URL				:	$URL: http://almscdc.swisslog.com/repo/SWPD/Development/BoxControlFramework/20_Release/trunk/01_Software/BCF/BCF/JumpStart/20_Product/10_App/10_Base/10_Lib/01_DUTs/ST_Base.TcDUT $
 *
 *	Purpose			:	Base framework structure
 *
 * ------------------------------------------------------------------------------------
 *	Copyright Swisslog [IP AG], Switzerland. All rights reserved.
 * 
 * ------------------------------------------------------------------------------------
 *	
 * 	Revision History: 
 *
 * 	VERSION			DATE			INITIALS			DESCRIPTION
 *	0.1				01.01.2001		swl					Example
 *
 **************************************************************************************)
STRUCT
	fbGetSystemTime	: GETSYSTEMTIME; // Get current system time
	VIR_Data		: ST_VIR_Data; // Visualization report values
	VIQ				: ST_ITC_VIQ; // ITC Message
	VIR_SEND_CLOCK	: UDINT := 3; // Send clock for VIR Report [s]
	CM				: ST_CM_Base;	/// Data Aquisition Variables Staorage and Settings // CM inside base 
END_STRUCT
END_TYPE

// ---- 20_Product/10_BCF/10_Base/01_DUTs/ST_CM_Base.TcDUT
TYPE ST_CM_Base :
(**************************************************************************************
 * 	Application		:	BoxControl Framework
 *	Revision		:	$Revision: 404529 $
 *	Revision date	:	$Date: 2018-04-23 08:21:38 +0200 (Mo., 23 Apr 2018) $
 *	Last changed by	:	$Author: b7bolm $
 *	URL				:	$URL: http://almscdc.swisslog.com/repo/SWPD/Development/BoxControlFramework/20_Release/trunk/01_Software/BCF/BCF/JumpStart/20_Product/10_App/10_Base/10_Lib/01_DUTs/ST_CM_Base.TcDUT $
 *
 *	Purpose			:	Base Structure for Condition monitoring 					
 *
 *
 * ------------------------------------------------------------------------------------
 *	Copyright Swisslog [IP AG], Switzerland. All rights reserved.
 * 
 * ------------------------------------------------------------------------------------
 *	
 * 	Revision History: 
 *
 * 	VERSION			DATE			INITIALS			DESCRIPTION
 *	0.1				01.01.2001		swl					Example
 *
 **************************************************************************************)	
STRUCT
	nCurrentTime 	: ULINT; // Current DC-Time of the PLC-Task
	DAQ				: ST_ITC_DAQ;	/// ITC Message
	GDQ				: ST_ITC_GDQ;	/// ITC Message
	Data			: ARRAY[E_CM_Index.E_BEGIN_VARIABLE+1..E_CM_Index.E_END_VARIABLE-1] OF ST_CM_GeneralData; //Process Data used by Condiition Monitoring Method 
	Settings		: ARRAY[E_CM_Index.E_BEGIN_VARIABLE+1..E_CM_Index.E_END_VARIABLE-1] OF ST_CM_Settings; //Settings Data set by Telegram/User
END_STRUCT
END_TYPE

// ---- 20_Product/10_BCF/10_Base/01_DUTs/ST_CM_GeneralData.TcDUT
TYPE ST_CM_GeneralData :
(**************************************************************************************
 * 	Application		:	BoxControl Framework
 *	Revision		:	$Revision: 404529 $
 *	Revision date	:	$Date: 2018-04-23 08:21:38 +0200 (Mo., 23 Apr 2018) $
 *	Last changed by	:	$Author: b7bolm $
 *	URL				:	$URL: http://almscdc.swisslog.com/repo/SWPD/Development/BoxControlFramework/20_Release/trunk/01_Software/BCF/BCF/JumpStart/20_Product/10_App/10_Base/10_Lib/01_DUTs/ST_CM_GeneralData.TcDUT $
 *
 *	Purpose			:	General Process data for Condition monitoring 					
 *
 *
 * ------------------------------------------------------------------------------------
 *	Copyright Swisslog [IP AG], Switzerland. All rights reserved.
 * 
 * ------------------------------------------------------------------------------------
 *	
 * 	Revision History: 
 *
 * 	VERSION			DATE			INITIALS			DESCRIPTION
 *	0.1				01.01.2001		swl					Example
 *
 **************************************************************************************)	
STRUCT
	Position			: STRING(Conveyor.POSITION_STRINGLENGTH);// PositionName MM-000-0000-000
	LoggingActive		: BOOL; //Logging is active 
	WriteIdx			: INT; //Write index
	SampleTimer			: ULINT; //Sample Timer 
	MaxReportTimer		: ULINT; // Maimum Report Timer 
	PreviousValue		: UDINT; // Last Value Logged 
	eMode				: E_CM_Mode; //Mode Selection 
	Sequence			: INT; //sequnce used for the Data log 
	Buffer				: ARRAY[0..System.CM_MAX_NUMBER_Of_ENTRIES] OF ST_CM_LOG; //Storage Buffer 
END_STRUCT
END_TYPE

// ---- 20_Product/10_BCF/10_Base/01_DUTs/ST_CM_Log.TcDUT
TYPE ST_CM_Log :
(**************************************************************************************
 * 	Application		:	BoxControl Framework
 *	Revision		:	$Revision: 404529 $
 *	Revision date	:	$Date: 2018-04-23 08:21:38 +0200 (Mo., 23 Apr 2018) $
 *	Last changed by	:	$Author: b7bolm $
 *	URL				:	$URL: http://almscdc.swisslog.com/repo/SWPD/Development/BoxControlFramework/20_Release/trunk/01_Software/BCF/BCF/JumpStart/20_Product/10_App/10_Base/10_Lib/01_DUTs/ST_CM_Log.TcDUT $
 *
 *	Purpose			:	Structure of Data Buffer for Condition monitoring 					
 *
 *
 * ------------------------------------------------------------------------------------
 *	Copyright Swisslog [IP AG], Switzerland. All rights reserved.
 * 
 * ------------------------------------------------------------------------------------
 *	
 * 	Revision History: 
 *
 * 	VERSION			DATE			INITIALS			DESCRIPTION
 *	0.1				01.01.2001		swl					Example
 *
 **************************************************************************************)	
STRUCT
	Value		: STRING(Conveyor.GATHERED_DATA_VALUE); //Captured Value
	TimeStamp	: STRING(System.CM_TIMESTAMP_MS_STRINGLENGTH); //Time Stamp
	Sequence	: INT; // Storage Sequence 
END_STRUCT
END_TYPE

// ---- 20_Product/10_BCF/10_Base/01_DUTs/ST_CM_Settings.TcDUT
TYPE ST_CM_Settings :
(**************************************************************************************
 * 	Application		:	BoxControl Framework
 *	Revision		:	$Revision: 404529 $
 *	Revision date	:	$Date: 2018-04-23 08:21:38 +0200 (Mo., 23 Apr 2018) $
 *	Last changed by	:	$Author: b7bolm $
 *	URL				:	$URL: http://almscdc.swisslog.com/repo/SWPD/Development/BoxControlFramework/20_Release/trunk/01_Software/BCF/BCF/JumpStart/20_Product/10_App/10_Base/10_Lib/01_DUTs/ST_CM_Settings.TcDUT $
 *
 *	Purpose			:	Condition Monitor Variable Settings Set via Telegram					
 *
 *
 * ------------------------------------------------------------------------------------
 *	Copyright Swisslog [IP AG], Switzerland. All rights reserved.
 * 
 * ------------------------------------------------------------------------------------
 *	
 * 	Revision History: 
 *
 * 	VERSION			DATE			INITIALS			DESCRIPTION
 *	0.1				01.01.2001		swl					Example
 *
 **************************************************************************************)	
STRUCT
	mVariableName		: STRING(System.CM_VARIABLENAME_STRINGLENGTH); //Variable Name 
	MaxReportTime		: TIME; // Maximum RpertTime hh:mm:ss	Default:’00:00:00’ = off
	SampleTime			: TIME; // Sample Report Time hh:mm:ss.SSS
	Threshold			: INT;  // Threshold – Minimum value change to capture a new value
	Option				: BOOL; //  Self-reset = FALSE , Reset forbidden:= True
	Enable				: BOOL; // Enable Logging 
	ErrorCode			: INT;  // Error Code 
END_STRUCT
END_TYPE

// ---- 20_Product/10_BCF/10_Base/01_DUTs/ST_ISR_Table.TcDUT
TYPE ST_ISR_Table :
(**************************************************************************************
 * 	Application		:	BoxControl Framework
 *	Revision		:	$Revision: 404529 $
 *	Revision date	:	$Date: 2018-04-23 08:21:38 +0200 (Mo., 23 Apr 2018) $
 *	Last changed by	:	$Author: b7bolm $
 *	URL				:	$URL: http://almscdc.swisslog.com/repo/SWPD/Development/BoxControlFramework/20_Release/trunk/01_Software/BCF/BCF/JumpStart/20_Product/10_App/10_Base/10_Lib/01_DUTs/ST_ISR_Table.TcDUT $
 *
 *	Purpose			:	ISR Signal Number
 *
 * ------------------------------------------------------------------------------------
 *	Copyright Swisslog [IP AG], Switzerland. All rights reserved.
 * 
 * ------------------------------------------------------------------------------------
 *	
 * 	Revision History: 
 *
 * 	VERSION			DATE			INITIALS			DESCRIPTION
 *	0.1				01.01.2001		swl					Example
 *
 **************************************************************************************)
STRUCT
	SignalNumber		: ARRAY [1..NUMBER_OF_ISR_SIGNALS] OF BOOL; // Array of Signal Numbers
END_STRUCT
END_TYPE

// ---- 20_Product/10_BCF/10_Base/01_DUTs/ST_PointerSet.TcDUT
TYPE ST_PointerSet :
STRUCT
	pAdr	: PVOID;
	Len		: UDINT;
END_STRUCT
END_TYPE

// ---- 20_Product/10_BCF/10_Base/01_DUTs/ST_PositionInfo.TcDUT
TYPE ST_PositionInfo :
(**************************************************************************************
 * 	Application		:	BoxControl Framework
 *	Revision		:	$Revision: 404529 $
 *	Revision date	:	$Date: 2018-04-23 08:21:38 +0200 (Mo., 23 Apr 2018) $
 *	Last changed by	:	$Author: b7bolm $
 *	URL				:	$URL: http://almscdc.swisslog.com/repo/SWPD/Development/BoxControlFramework/20_Release/trunk/01_Software/BCF/BCF/JumpStart/20_Product/10_App/10_Base/10_Lib/01_DUTs/ST_PositionInfo.TcDUT $
 *
 *	Purpose			:	Position info
 *
 * ------------------------------------------------------------------------------------
 *	Copyright Swisslog [IP AG], Switzerland. All rights reserved.
 * 
 * ------------------------------------------------------------------------------------
 *	
 * 	Revision History: 
 *
 * 	VERSION			DATE			INITIALS			DESCRIPTION
 *	0.1				01.01.2001		swl					Example
 *
 **************************************************************************************)	
STRUCT
	SystemReady		: BOOL; // Subsystem ready
	E_Stopped		: BOOL; // Emergency stop active
	Maintenance		: BOOL; // Maintenance active
END_STRUCT
END_TYPE

// ---- 20_Product/10_BCF/10_Base/01_DUTs/ST_PositionState.TcDUT
TYPE ST_PositionState :
(**************************************************************************************
 * 	Application		:	BoxControl Framework
 *	Revision		:	$Revision: 404529 $
 *	Revision date	:	$Date: 2018-04-23 08:21:38 +0200 (Mo., 23 Apr 2018) $
 *	Last changed by	:	$Author: b7bolm $
 *	URL				:	$URL: http://almscdc.swisslog.com/repo/SWPD/Development/BoxControlFramework/20_Release/trunk/01_Software/BCF/BCF/JumpStart/20_Product/10_App/10_Base/10_Lib/01_DUTs/ST_PositionState.TcDUT $
 *
 *	Purpose			:	Position state
 *
 * ------------------------------------------------------------------------------------
 *	Copyright Swisslog [IP AG], Switzerland. All rights reserved.
 * 
 * ------------------------------------------------------------------------------------
 *	
 * 	Revision History: 
 *
 * 	VERSION			DATE			INITIALS			DESCRIPTION
 *	0.1				01.01.2001		swl					Example
 *
 **************************************************************************************)	
STRUCT
	eMode			: E_PositionMode; // Mode of the group 
	eState 			: E_PositionState; // State of the group 
	eLastState		: E_PositionState; // Previous state of the group 
	Info			: ST_PositionInfo; // Position info
	InitRelease		: ST_InitRelease; // Release to init 
END_STRUCT
END_TYPE

// ---- 20_Product/10_BCF/10_Base/01_DUTs/ST_SDI_Table.TcDUT
TYPE ST_SDI_Table :
(**************************************************************************************
 * 	Application		:	BoxControl Framework
 *	Revision		:	$Revision: 404529 $
 *	Revision date	:	$Date: 2018-04-23 08:21:38 +0200 (Mo., 23 Apr 2018) $
 *	Last changed by	:	$Author: b7bolm $
 *	URL				:	$URL: http://almscdc.swisslog.com/repo/SWPD/Development/BoxControlFramework/20_Release/trunk/01_Software/BCF/BCF/JumpStart/20_Product/10_App/10_Base/10_Lib/01_DUTs/ST_SDI_Table.TcDUT $
 *
 *	Purpose			:	SDI table
 *
 * ------------------------------------------------------------------------------------
 *	Copyright Swisslog [IP AG], Switzerland. All rights reserved.
 * 
 * ------------------------------------------------------------------------------------
 *	
 * 	Revision History: 
 *
 * 	VERSION			DATE			INITIALS			DESCRIPTION
 *	0.1				01.01.2001		swl					Example
 *
 **************************************************************************************)
STRUCT
	Enabled			: BOOL; // SDI signal enabled
	State			: BOOL; // Current State of the SDI 
	LastState		: BOOL; // The last state of the SDI 
END_STRUCT
END_TYPE

// ---- 20_Product/10_BCF/10_Base/01_DUTs/ST_VIR_Data.TcDUT
TYPE ST_VIR_Data :
(**************************************************************************************
 * 	Application		:	BoxControl Framework
 *	Revision		:	$Revision: 404529 $
 *	Revision date	:	$Date: 2018-04-23 08:21:38 +0200 (Mo., 23 Apr 2018) $
 *	Last changed by	:	$Author: b7bolm $
 *	URL				:	$URL: http://almscdc.swisslog.com/repo/SWPD/Development/BoxControlFramework/20_Release/trunk/01_Software/BCF/BCF/JumpStart/20_Product/10_App/10_Base/10_Lib/01_DUTs/ST_VIR_Data.TcDUT $
 *
 *	Purpose			:	Visualization report structure
 *
 *
 * ------------------------------------------------------------------------------------
 *	Copyright Swisslog [IP AG], Switzerland. All rights reserved.
 * 
 * ------------------------------------------------------------------------------------
 *	
 * 	Revision History: 
 *
 * 	VERSION			DATE			INITIALS			DESCRIPTION
 *	0.1				01.01.2001		swl					Example
 *
 **************************************************************************************)
STRUCT
	SendingAllowed			: BOOL; // Its allowed to send a new report
	Overflow				: BOOL; // Overflow detected
	TimeStep				: UDINT; // Desired time step
	NextSendTimeStamp		: UDINT; // Next possible timestamp
	ChangeDetected			: BOOL; // Change detected
	NumberOfUsedKeys	 	: INT; // Number of monitored keys
	Data					: ARRAY [1..System.NUMBER_OF_KEYVALUE_PAIRS_VIR] OF ST_ITC_VIR_SET; // Valid data
	PrepData				: ARRAY [1..System.NUMBER_OF_KEYVALUE_PAIRS_VIR] OF ST_ITC_VIR_SET; // Preparation for sending report
END_STRUCT
END_TYPE

// ---- 20_Product/10_BCF/10_Base/10_StateMachine/A_InstancePath.TcDUT
// alias for instance path string
TYPE
  A_InstancePath : STRING[255];
END_TYPE

// ---- 20_Product/10_BCF/10_Base/10_StateMachine/A_StateText.TcDUT
// alias for a state text for FB_StateMachine
TYPE
  A_StateText    : STRING[31];
END_TYPE

// ---- 20_Product/10_BCF/10_Base/11_Com/02_Timings/E_BlinkFrequencies.TcDUT
// blink frequencies for F_GetBlinkCycle
{attribute 'qualified_only'}
{attribute 'strict'}
TYPE E_BlinkFrequencies:

(**************************************************************************************
 * 	Application		:	BoxControl Framework
 *	Revision		  :	$Revision: 461868 $
 *	Revision date	:	$Date: 1979-01-09 14:35:13 +0200 (Di., 09 Jan 1979) $
 *	Last changed by	:	$Author: b7lipim $
 *	URL				:	$URL: http://almscdc.swisslog.com/repo/SWPD/Development/BoxControlFramework/20_Release/branches/R1.x/01_Software/BCF/BCF/JumpStart/20_Product/10_BCF/10_Base/11_Com/12_DebugMsg/00_GVLs/DebugTextBlocks.TcGVL $
 *
 * ------------------------------------------------------------------------------------
 *	Copyright Swisslog [IP AG], Switzerland. All rights reserved.
 * 
 * ------------------------------------------------------------------------------------
 *	
 * 	Revision History: 
 *
 * VERSION DATE         INITIALS     DESCRIPTION
 * 0.0     DD.MM.YYYY   (name)       (explain customized modifications)
 *
 **************************************************************************************)

(
  Off          := 2#0000_0000_0000_0000,     // off
  //----------------------------------------------------------------------
//Hertz_500    := 2#0000_0000_0000_0001,     // 500Hz
//Hertz_250    := 2#0000_0000_0000_0010,     // 250Hz
//Hertz_125    := 2#0000_0000_0000_0100,     // 125Hz
//Hertz_64     := 2#0000_0000_0000_1000,     //  64Hz    ( 62.5 )
//Hertz_32     := 2#0000_0000_0001_0000,     //  32Hz    ( 31.25 )
//Hertz_16     := 2#0000_0000_0010_0000,     //  16Hz    ( 15.625 )
  Hertz_8      := 2#0000_0000_0100_0000,     //   8Hz    (  7.8125 )
  Hertz_4      := 2#0000_0000_1000_0000,     //   4Hz    (  3.90625 ) 
  Hertz_2      := 2#0000_0001_0000_0000,     //   2Hz    (  1.953125 )
  Hertz_1      := 2#0000_0010_0000_0000,     //   1Hz    (  0.9765625 )
  Hertz_0_5    := 2#0000_0100_0000_0000,     // 1/2 Hz   (  0.48828125 )
  Hertz_0_25   := 2#0000_1000_0000_0000,     // 1/4 Hz   (  0.244140625 )
  Hertz_0_125  := 2#0001_0000_0000_0000,     // 1/8 Hz   (  0.1220703125 )
  //----------------------------------------------------------------------
  On           := 2#1111_1111_1111_1111      // on
) DWORD;
END_TYPE

// ---- 20_Product/10_BCF/10_Base/11_Com/12_DebugMsg/01_DUTs/E_DebugMsgType.TcDUT
{attribute 'qualified_only'}
{attribute 'strict'}
{attribute 'to_string'}
TYPE E_DebugMsgType :
(**************************************************************************************
 * 	Application		:	BoxControl Framework
 *	Revision		:	$Revision: 404529 $
 *	Revision date	:	$Date: 2018-04-23 08:21:38 +0200 (Mo., 23 Apr 2018) $
 *	Last changed by	:	$Author: b7bolm $
 *	URL				:	$URL: http://almscdc.swisslog.com/repo/SWPD/Development/BoxControlFramework/20_Release/trunk/01_Software/BCF/BCF/JumpStart/20_Product/10_App/11_Com/10_Lib/01_DUTs/E_DebugMsgType.TcDUT $
 *
 *	Purpose			:	Debug message type
 *
 * ------------------------------------------------------------------------------------
 *	Copyright Swisslog [IP AG], Switzerland. All rights reserved.
 * 
 * ------------------------------------------------------------------------------------
 *	
 * 	Revision History: 
 *
 * VERSION DATE         INITIALS     DESCRIPTION
 * 0.0     DD.MM.YYYY   (name)       (explain customized modifications)
 *
 **************************************************************************************)	
(
	INFO ,
	WARNING,
	ERROR
);
END_TYPE

// ---- 20_Product/10_BCF/10_Base/11_Com/12_DebugMsg/01_DUTs/ST_CFG_DebugMsgManager.TcDUT
TYPE ST_CFG_DebugMsgManager :
STRUCT
	TCP_Driver		: ST_CFG_TcpDriver;
	SystemNumber	: INT;
END_STRUCT
END_TYPE

// ---- 20_Product/10_BCF/11_Conv/10_Base/01_DUTs/E_ErrorConv.TcDUT
TYPE E_ErrorConv :
(**************************************************************************************
 * 	Application		:	BoxControl Framework
 *	Revision		:	$Revision: 404529 $
 *	Revision date	:	$Date: 2018-04-23 08:21:38 +0200 (Mo., 23 Apr 2018) $
 *	Last changed by	:	$Author: b7bolm $
 *	URL				:	$URL: http://almscdc.swisslog.com/repo/SWPD/Development/BoxControlFramework/20_Release/trunk/01_Software/BCF/BCF/JumpStart/20_Product/10_App/10_Base/10_Lib/10_Conv/01_DUTs/E_ErrorConv.TcDUT $
 *
 *	Purpose			:	Basic conveyor error list. Limited range 0-999.
 *						All codes have to be set to a value!
 *
 * ------------------------------------------------------------------------------------
 *	Copyright Swisslog [IP AG], Switzerland. All rights reserved.
 * 
 * ------------------------------------------------------------------------------------
 *	
 * 	Revision History: 
 *
 * 	VERSION			DATE			INITIALS			DESCRIPTION
 *	0.1				01.01.2001		swl					Example
 *
 *************************************************************************************)
(
  NO_ERROR_CODE                             := 0000, // No error 


  (*-------------------------------------------------------------
    IPC Hardware / System				
   -------------------------------------------------------------*)
  OVER_TEMPEREATURE_CPU                     := 0001, // Temperature limit CPU exceeded 
  OVER_TEMPEREATURE_MOTHERBOARD             := 0002, // Temperature limit motherboard exceeded 
  FAN_ERROR_CPU                             := 0003, // Fan speed is zero 
  CPU_OVERLOAD                              := 0004, // CPU usage limit exceeded
  IPC_EVENT_FASTSTOP                        := 0005, // FastStop because of an event in the Subsystem status 
  IPC_EVENT_SOFTSTOP                        := 0006, // SoftStop because of an event in the Subsystem status 


  (*-------------------------------------------------------------
    Communication	        			
  -------------------------------------------------------------*)
  CONNECTION_ERROR                          := 0020, // General connection error
  CONNECTION_ERROR_TO_AM                    := 0021, // Connection error to AM 
  CONNECTION_ERROR_TO_SPOC                  := 0022, // Connection error to SPOC 
  CONNECTION_ERROR_TO_EXTERNAL_INTERFACE    := 0023, // Connection error to external interface e.g. MLC 
  CONNECTION_ERROR_DEVICE                   := 0024, // Connection error to external device e.g. scale, printer


  (* -------------------------------------------------------------
    Communication MFCS					
  --------------------------------------------------------------*)
  AM_BUFFER_OVERFLOW                        := 0040, // Communication buffer to AM overflow
  WRONG_VALUE                               := 0041, // A wrong value in the telegram 
  DELETE_TU_DATA_NOT_POSSIBLE               := 0042, // Del TU-Data not possible, TU-Data position is empty 
  JOB_STILL_ACTIVE                          := 0043, // Job was still active during deleting TU 
  SUBSYSTEMNUMBER_UNKNOWN                   := 0044, // Wrong or inexistent Subsystem number 
  GROUPNUMBER_UNKNOWN                       := 0045, // Wrong or inexistent group number 
  ELEMENTNUMBER_UNKNOWN                     := 0046, // Wrong or inexistent element number 
  FUNCTIONNUMBER_UNKNOWN                    := 0047, // Wrong or inexistent function number 
  ZONENUMBER_INVALID                        := 0048, // Zone number not valid
  ROBOT_ITC_CONFIG_INVALID                  := 0049, // Non robot function 


  (* -------------------------------------------------------------
    Fieldbus				
  --------------------------------------------------------------*)
  ETHERCAT_MASTER_ERROR                     := 0060, // EtherCAT master error 
  ETHERCAT_MASTER_TELEGRAM_LOST             := 0061, // EtherCAT master telegrams lost 
  ETHERCAT_SLAVE_ERROR                      := 0062, // No connection to EtherCAT slave 


  (*-------------------------------------------------------------
    Groups	        			
   -------------------------------------------------------------*)
  CONTROL_VOLTAGE                           := 0080, // Control voltage has failed 
  OVERCURRENT                               := 0081, // Over current 
  EMERGENCY_STOP                            := 0082, // Emergency stop activated 
  MAIN_CONTACTOR_OFF                        := 0083, // Main contactor failure 
  FIRE_ALARM                                := 0084, // Fire alarm 
  AIR_PRESSURE_LOW                          := 0085, // Air pressure to low 
  MAINTENANCE                               := 0086, // Maintenance activated 
  FST_STOP_AFTER_TIMEOUT                    := 0087, // Faststop from a timeout, no SoftStop is possible 


  (*-------------------------------------------------------------
    Fuses	        			
   -------------------------------------------------------------*)
  FUSE_FAN_CABINET                          := 0090, // Cabinet Fan Fuse triggered
  FUSE_24VDC                                := 0091, // 24VDC Fuse triggered
  FUSE_400VAC                               := 0092, // 400VAC Fuse triggered


  (* -------------------------------------------------------------
     Material Flow 				
   --------------------------------------------------------------*)
  TU_ID_WRONG                               := 0100, // TU-ID is wrong 
  ASSIGNMENT_ID_WRONG                       := 0101, // Assignment ID wrong
  NO_FREE_TU_DATA_SET                       := 0102, // No free TU-DataSet found 
  INDEX_MATCH_WITH_POSITION                 := 0103, // TU-DataIndex is allocated to another position 
  TU_DATA_SET_EMPTY_ZONE_OCCUPIED           := 0104, // TU data set empty, position occupied 
  TU_DATA_SET_OCCUPIED_ZONE_FREE            := 0105, // TU data set occupied, position free 
  EMPTY_TU_DATA_SET                         := 0106, // No TU data found in source position 
  DESTINATION_INVALID                       := 0107, // Destination is invalid, delivery impossible 
  TU_WRONG_ORIENTATION                      := 0108, // TU wrong orientation, turn TU in right orientation 
  TU_DATA_INDEX_NOT_FREE                    := 0109, // TU-data index is not free
  ID_WRONG                                  := 0110, // Neither TU_ID nor Assignement_ID specified
  WRONG_TU_DATA_INDEX_RECEIVED              := 0111, // Wrong TU data index.
  ROBOT_TASK_INDEX_WRONG                    := 0112, // Robot task index is wrong 
  TU_DATA_INDEX_FREE                        := 0113, // TU data index is free
  DESTINATION_NOT_REACHABLE                 := 0114, // Specified destination not reachable 	
  TU_DATA_SET_EMPTY_OF_RECEIVING_TU         := 0115, // TU Idx of receiving TU is 0
  TU_LEFT_SUBSYSTEM                         := 0116, // TU has left subsystem


  (* -------------------------------------------------------------
    Error Timeouts						
  --------------------------------------------------------------*)
  TIMEOUT                                   := 0120, // General timeout message
  TIMEOUT_TAKEOVER                          := 0121, // Timeout during takeover 
  TIMEOUT_HANDOVER                          := 0122, // Timeout during hadover 
  TIMEOUT_LIFTING                           := 0123, // Timeout during lifting 
  TIMEOUT_MOVEMENT                          := 0124, // Timeout during movement
  TIMEOUT_DEVICE                            := 0125, // Timeout device
  TIMEOUT_STRATEGY                          := 0126, // Timeout strategy
  TIMEOUT_COMMUNICATION                     := 0127, // Communication timeout


  (* -------------------------------------------------------------
    Sensors Errors						
  ---------------------------------------------------------------*)
  INCORRECT_SENSOR_SIGNAL                   := 0140, // Incorrect signal of the sensors 
  INCORRECT_ENCODER_VALUE                   := 0141, // Incorrect value of the encoder 
  LIMIT_SWITCH_ACTIVE                       := 0142, // Limit switch is activated 
  GAP_CHECK_ACTIVE                          := 0143, // Gap check active


  (* -------------------------------------------------------------
    Profile Control Units Errors 			        
  --------------------------------------------------------------*)
  SENSOR_FRONT_DEFECT                       := 0160, // Front transmitter defective 
  SENSOR_REAR_DEFECT                        := 0161, // Rear transmitter defective 
  SENSOR_LEFT_DEFECT                        := 0162, // Left transmitter defective 
  SENSOR_RIGHT_DEFECT                       := 0163, // Right transmitter defective 
  SENSOR_HEIGHT_DEFECT                      := 0164, // Height transmitter defective 
  SENSOR_WEIGHT_DEFECT                      := 0165, // Transmitter for weight measurement defective 
  SENSOR_TUNNEL_DEFECT                      := 0166, // Transmitter to check space for forks defective 
  SENSOR_RUNNER_DEFECT                      := 0167, // Shelf sensor transmitter defective 
  SCALE_NOT_READY                           := 0168, // Scale not ready 


